LIN {X 0,Y 467.855,Z 196.206,A -85,B 0,C 180,E1 -7560,E2 -7560} C_VEL
LIN {X 0,Y 467.817,Z 196.211,A -85,B 0,C 180,E1 -7562.583,E2 -7562.583} C_VEL
LIN {X 0,Y 467.706,Z 196.227,A -85,B 0,C 180,E1 -7566.038,E2 -7566.038} C_VEL
LIN {X 0,Y 467.66,Z 196.229,A -85,B 0,C 180,E1 -7568.643,E2 -7568.643} C_VEL
LIN {X 0,Y 467.66,Z 196.234,A -85,B 0,C 180,E1 -7572.145,E2 -7572.145} C_VEL
LIN {X 0,Y 467.616,Z 196.236,A -85,B 0,C 180,E1 -7575.696,E2 -7575.696} C_VEL
LIN {X 0,Y 467.622,Z 196.233,A -85,B 0,C 180,E1 -7579.308,E2 -7579.308} C_VEL
LIN {X 0,Y 467.537,Z 196.247,A -85,B 0,C 180,E1 -7582.074,E2 -7582.074} C_VEL
LIN {X 0,Y 467.562,Z 196.239,A -85,B 0,C 180,E1 -7584.89,E2 -7584.89} C_VEL
LIN {X 0,Y 467.549,Z 196.248,A -85,B 0,C 180,E1 -7587.774,E2 -7587.774} C_VEL
LIN {X 0,Y 467.568,Z 196.24,A -85,B 0,C 180,E1 -7591.044,E2 -7591.044} C_VEL
LIN {X 0,Y 467.579,Z 196.238,A -85,B 0,C 180,E1 -7594.24,E2 -7594.24} C_VEL
LIN {X 0,Y 467.545,Z 196.245,A -85,B 0,C 180,E1 -7597.185,E2 -7597.185} C_VEL
LIN {X 0,Y 467.56,Z 196.239,A -85,B 0,C 180,E1 -7600.267,E2 -7600.267} C_VEL
LIN {X 0,Y 467.547,Z 196.244,A -85,B 0,C 180,E1 -7603.746,E2 -7603.746} C_VEL
LIN {X 0,Y 467.547,Z 196.241,A -85,B 0,C 180,E1 -7606.254,E2 -7606.254} C_VEL
LIN {X 0,Y 467.559,Z 196.241,A -85,B 0,C 180,E1 -7609.733,E2 -7609.733} C_VEL
LIN {X 0,Y 467.545,Z 196.245,A -85,B 0,C 180,E1 -7612.815,E2 -7612.815} C_VEL
LIN {X 0,Y 467.578,Z 196.237,A -85,B 0,C 180,E1 -7615.76,E2 -7615.76} C_VEL
LIN {X 0,Y 467.55,Z 196.248,A -85,B 0,C 180,E1 -7618.959,E2 -7618.959} C_VEL
LIN {X 0,Y 467.613,Z 196.32,A -85,B 0,C 180,E1 -7622.23,E2 -7622.23} C_VEL
LIN {X 0,Y 470.285,Z 209.821,A -85,B 0,C 180,E1 -7624.555,E2 -7624.555} C_VEL
LIN {X 0,Y 469.734,Z 224.485,A -85,B 0,C 180,E1 -7626.874,E2 -7626.874} C_VEL
LIN {X 0,Y 468.948,Z 244.938,A -85,B 0,C 180,E1 -7630.065,E2 -7630.065} C_VEL
LIN {X 0,Y 468.232,Z 264.095,A -85,B 0,C 180,E1 -7633.005,E2 -7633.005} C_VEL
LIN {X 0,Y 471.04,Z 286.598,A -85,B 0,C 180,E1 -7633.47,E2 -7633.47} C_VEL
LIN {X 0,Y 470.274,Z 373.12,A -85,B 0,C 180,E1 -7634.867,E2 -7634.867} C_VEL
LIN {X 0,Y 469.84,Z 386.276,A -85,B 0,C 180,E1 -7635.24,E2 -7635.24} C_VEL
LIN {X 0,Y 469.395,Z 399.568,A -85,B 0,C 180,E1 -7635.808,E2 -7635.808} C_VEL
LIN {X 0,Y 468.88,Z 410.763,A -85,B 0,C 180,E1 -7636.455,E2 -7636.455} C_VEL
LIN {X 0,Y 468.297,Z 422.997,A -85,B 0,C 180,E1 -7637.369,E2 -7637.369} C_VEL
LIN {X 0,Y 467.927,Z 434.003,A -85,B 0,C 180,E1 -7638.411,E2 -7638.411} C_VEL
LIN {X 0,Y 467.422,Z 444.065,A -85,B 0,C 180,E1 -7639.605,E2 -7639.605} C_VEL
LIN {X 0,Y 467.139,Z 452.942,A -85,B 0,C 180,E1 -7640.911,E2 -7640.911} C_VEL
LIN {X 0,Y 466.928,Z 460.016,A -85,B 0,C 180,E1 -7642.214,E2 -7642.214} C_VEL
LIN {X 0,Y 466.829,Z 465.703,A -85,B 0,C 180,E1 -7643.523,E2 -7643.523} C_VEL
LIN {X 0,Y 466.765,Z 470.118,A -85,B 0,C 180,E1 -7644.817,E2 -7644.817} C_VEL
LIN {X 0,Y 466.697,Z 472.456,A -85,B 0,C 180,E1 -7645.682,E2 -7645.682} C_VEL
LIN {X 0,Y 466.786,Z 474.366,A -85,B 0,C 180,E1 -7646.547,E2 -7646.547} C_VEL
LIN {X 0,Y 466.787,Z 475.795,A -85,B 0,C 180,E1 -7647.411,E2 -7647.411} C_VEL
LIN {X 0,Y 466.705,Z 476.796,A -85,B 0,C 180,E1 -7648.274,E2 -7648.274} C_VEL
LIN {X 0,Y 466.651,Z 477.608,A -85,B 0,C 180,E1 -7650,E2 -7650} C_VEL
LIN {X 0,Y 466.653,Z 477.372,A -85,B 0,C 180,E1 -7650.863,E2 -7650.863} C_VEL
LIN {X 0,Y 466.706,Z 476.732,A -85,B 0,C 180,E1 -7651.726,E2 -7651.726} C_VEL
LIN {X 0,Y 466.79,Z 475.696,A -85,B 0,C 180,E1 -7652.589,E2 -7652.589} C_VEL
LIN {X 0,Y 466.8,Z 474.243,A -85,B 0,C 180,E1 -7653.452,E2 -7653.452} C_VEL
LIN {X 0,Y 466.707,Z 471.192,A -85,B 0,C 180,E1 -7654.751,E2 -7654.751} C_VEL
LIN {X 0,Y 466.747,Z 467.084,A -85,B 0,C 180,E1 -7656.05,E2 -7656.05} C_VEL
LIN {X 0,Y 466.903,Z 460.778,A -85,B 0,C 180,E1 -7657.568,E2 -7657.568} C_VEL
LIN {X 0,Y 467.063,Z 453.902,A -85,B 0,C 180,E1 -7658.872,E2 -7658.872} C_VEL
LIN {X 0,Y 467.351,Z 445.386,A -85,B 0,C 180,E1 -7660.177,E2 -7660.177} C_VEL
LIN {X 0,Y 467.801,Z 436.641,A -85,B 0,C 180,E1 -7661.262,E2 -7661.262} C_VEL
LIN {X 0,Y 468.157,Z 426.895,A -85,B 0,C 180,E1 -7662.257,E2 -7662.257} C_VEL
LIN {X 0,Y 468.706,Z 415.217,A -85,B 0,C 180,E1 -7663.218,E2 -7663.218} C_VEL
LIN {X 0,Y 469.206,Z 403.457,A -85,B 0,C 180,E1 -7663.977,E2 -7663.977} C_VEL
LIN {X 0,Y 469.675,Z 391.29,A -85,B 0,C 180,E1 -7664.57,E2 -7664.57} C_VEL
LIN {X 0,Y 470.121,Z 378.153,A -85,B 0,C 180,E1 -7665.027,E2 -7665.027} C_VEL
LIN {X 0,Y 470.426,Z 365.707,A -85,B 0,C 180,E1 -7665.294,E2 -7665.294} C_VEL
LIN {X 0,Y 470.993,Z 284.423,A -85,B 0,C 180,E1 -7666.606,E2 -7666.606} C_VEL
LIN {X 0,Y 468.16,Z 262.297,A -85,B 0,C 180,E1 -7667.094,E2 -7667.094} C_VEL
LIN {X 0,Y 468.769,Z 243.285,A -85,B 0,C 180,E1 -7669.942,E2 -7669.942} C_VEL
LIN {X 0,Y 469.439,Z 222.22,A -85,B 0,C 180,E1 -7673.141,E2 -7673.141} C_VEL
LIN {X 0,Y 469.889,Z 208.581,A -85,B 0,C 180,E1 -7675.231,E2 -7675.231} C_VEL
LIN {X 0,Y 467.93,Z 197.894,A -85,B 0,C 180,E1 -7677,E2 -7677} C_VEL
LIN {X 0,Y 467.605,Z 196.242,A -85,B 0,C 180,E1 -7677.29,E2 -7677.29} C_VEL
LIN {X 0,Y 467.564,Z 196.247,A -85,B 0,C 180,E1 -7680.734,E2 -7680.734} C_VEL
LIN {X 0,Y 467.57,Z 196.241,A -85,B 0,C 180,E1 -7683.789,E2 -7683.789} C_VEL
LIN {X 0,Y 467.524,Z 196.25,A -85,B 0,C 180,E1 -7686.962,E2 -7686.962} C_VEL
LIN {X 0,Y 467.564,Z 196.24,A -85,B 0,C 180,E1 -7689.951,E2 -7689.951} C_VEL
LIN {X 0,Y 467.56,Z 196.245,A -85,B 0,C 180,E1 -7692.563,E2 -7692.563} C_VEL
LIN {X 0,Y 467.565,Z 196.241,A -85,B 0,C 180,E1 -7695.052,E2 -7695.052} C_VEL
LIN {X 0,Y 467.567,Z 196.245,A -85,B 0,C 180,E1 -7698.596,E2 -7698.596} C_VEL
LIN {X 0,Y 467.561,Z 196.243,A -85,B 0,C 180,E1 -7701.955,E2 -7701.955} C_VEL
LIN {X 0,Y 467.562,Z 196.239,A -85,B 0,C 180,E1 -7705.167,E2 -7705.167} C_VEL
LIN {X 0,Y 467.582,Z 196.242,A -85,B 0,C 180,E1 -7708.26,E2 -7708.26} C_VEL
LIN {X 0,Y 467.555,Z 196.24,A -85,B 0,C 180,E1 -7711.249,E2 -7711.249} C_VEL
LIN {X 0,Y 467.583,Z 196.242,A -85,B 0,C 180,E1 -7714.158,E2 -7714.158} C_VEL
LIN {X 0,Y 467.576,Z 196.237,A -85,B 0,C 180,E1 -7716.996,E2 -7716.996} C_VEL
LIN {X 0,Y 467.622,Z 196.236,A -85,B 0,C 180,E1 -7719.777,E2 -7719.777} C_VEL
LIN {X 0,Y 467.594,Z 196.235,A -85,B 0,C 180,E1 -7722.506,E2 -7722.506} C_VEL
LIN {X 0,Y 467.601,Z 196.236,A -85,B 0,C 180,E1 -7725.196,E2 -7725.196} C_VEL
LIN {X 0,Y 467.656,Z 196.231,A -85,B 0,C 180,E1 -7727.854,E2 -7727.854} C_VEL
LIN {X 0,Y 467.68,Z 196.228,A -85,B 0,C 180,E1 -7731.357,E2 -7731.357} C_VEL
LIN {X 0,Y 467.735,Z 196.221,A -85,B 0,C 180,E1 -7733.962,E2 -7733.962} C_VEL
LIN {X 0,Y 467.859,Z 196.21,A -85,B 0,C 180,E1 -7737.417,E2 -7737.417} C_VEL
LIN {X 0,Y 467.882,Z 196.202,A -85,B 0,C 180,E1 -7740,E2 -7740} C_VEL
LIN {X 0,Y 467.859,Z 196.205,A -85,B 0,C 180,E1 -7742.583,E2 -7742.583} C_VEL
LIN {X 0,Y 467.724,Z 196.22,A -85,B 0,C 180,E1 -7746.038,E2 -7746.038} C_VEL
LIN {X 0,Y 467.66,Z 196.233,A -85,B 0,C 180,E1 -7749.515,E2 -7749.515} C_VEL
LIN {X 0,Y 467.654,Z 196.233,A -85,B 0,C 180,E1 -7752.358,E2 -7752.358} C_VEL
LIN {X 0,Y 467.649,Z 196.233,A -85,B 0,C 180,E1 -7755.885,E2 -7755.885} C_VEL
LIN {X 0,Y 467.628,Z 196.237,A -85,B 0,C 180,E1 -7759.308,E2 -7759.308} C_VEL
LIN {X 0,Y 467.664,Z 196.309,A -85,B 0,C 180,E1 -7760.393,E2 -7760.393} C_VEL
LIN {X 0,Y 468.236,Z 199.2,A -85,B 0,C 180,E1 -7760.97,E2 -7760.97} C_VEL
LIN {X 0,Y 470.703,Z 207.594,A -85,B 0,C 180,E1 -7761.225,E2 -7761.225} C_VEL
LIN {X 0,Y 471.622,Z 212.53,A -85,B 0,C 180,E1 -7761.345,E2 -7761.345} C_VEL
LIN {X 0,Y 470.638,Z 307.216,A -85,B 0,C 180,E1 -7762.904,E2 -7762.904} C_VEL
LIN {X 0,Y 470.441,Z 320.163,A -85,B 0,C 180,E1 -7763.292,E2 -7763.292} C_VEL
LIN {X 0,Y 470.108,Z 333.13,A -85,B 0,C 180,E1 -7763.864,E2 -7763.864} C_VEL
LIN {X 0,Y 469.705,Z 344.998,A -85,B 0,C 180,E1 -7764.58,E2 -7764.58} C_VEL
LIN {X 0,Y 469.182,Z 356.975,A -85,B 0,C 180,E1 -7765.509,E2 -7765.509} C_VEL
LIN {X 0,Y 468.735,Z 367.183,A -85,B 0,C 180,E1 -7766.516,E2 -7766.516} C_VEL
LIN {X 0,Y 468.292,Z 377.042,A -85,B 0,C 180,E1 -7767.726,E2 -7767.726} C_VEL
LIN {X 0,Y 467.817,Z 385.718,A -85,B 0,C 180,E1 -7769.055,E2 -7769.055} C_VEL
LIN {X 0,Y 467.469,Z 393.089,A -85,B 0,C 180,E1 -7770.491,E2 -7770.491} C_VEL
LIN {X 0,Y 467.257,Z 398.252,A -85,B 0,C 180,E1 -7771.765,E2 -7771.765} C_VEL
LIN {X 0,Y 467.021,Z 403.063,A -85,B 0,C 180,E1 -7773.317,E2 -7773.317} C_VEL
LIN {X 0,Y 466.843,Z 406.389,A -85,B 0,C 180,E1 -7774.894,E2 -7774.894} C_VEL
LIN {X 0,Y 466.758,Z 407.877,A -85,B 0,C 180,E1 -7775.96,E2 -7775.96} C_VEL
LIN {X 0,Y 466.714,Z 408.708,A -85,B 0,C 180,E1 -7777.051,E2 -7777.051} C_VEL
LIN {X 0,Y 466.711,Z 408.872,A -85,B 0,C 180,E1 -7778.46,E2 -7778.46} C_VEL
LIN {X 0,Y 466.727,Z 408.015,A -85,B 0,C 180,E1 -7779.829,E2 -7779.829} C_VEL
LIN {X 0,Y 466.827,Z 405.646,A -85,B 0,C 180,E1 -7781.484,E2 -7781.484} C_VEL
LIN {X 0,Y 467.062,Z 401.512,A -85,B 0,C 180,E1 -7783.189,E2 -7783.189} C_VEL
LIN {X 0,Y 467.269,Z 396.435,A -85,B 0,C 180,E1 -7784.68,E2 -7784.68} C_VEL
LIN {X 0,Y 467.486,Z 389.628,A -85,B 0,C 180,E1 -7786.188,E2 -7786.188} C_VEL
LIN {X 0,Y 467.855,Z 382.299,A -85,B 0,C 180,E1 -7787.47,E2 -7787.47} C_VEL
LIN {X 0,Y 468.317,Z 373.785,A -85,B 0,C 180,E1 -7788.677,E2 -7788.677} C_VEL
LIN {X 0,Y 468.706,Z 364.825,A -85,B 0,C 180,E1 -7789.712,E2 -7789.712} C_VEL
LIN {X 0,Y 469.123,Z 353.914,A -85,B 0,C 180,E1 -7790.732,E2 -7790.732} C_VEL
LIN {X 0,Y 469.633,Z 342.07,A -85,B 0,C 180,E1 -7791.608,E2 -7791.608} C_VEL
LIN {X 0,Y 470.004,Z 330.609,A -85,B 0,C 180,E1 -7792.26,E2 -7792.26} C_VEL
LIN {X 0,Y 470.257,Z 317.363,A -85,B 0,C 180,E1 -7792.819,E2 -7792.819} C_VEL
LIN {X 0,Y 470.415,Z 311.813,A -85,B 0,C 180,E1 -7792.992,E2 -7792.992} C_VEL
LIN {X 0,Y 469.918,Z 306.092,A -85,B 0,C 180,E1 -7793.162,E2 -7793.162} C_VEL
LIN {X 0,Y 464.426,Z 287.452,A -85,B 0,C 180,E1 -7793.665,E2 -7793.665} C_VEL
LIN {X 0,Y 463.873,Z 281.633,A -85,B 0,C 180,E1 -7793.774,E2 -7793.774} C_VEL
LIN {X 0,Y 464.524,Z 212.332,A -85,B 0,C 180,E1 -7794.906,E2 -7794.906} C_VEL
LIN {X 0,Y 462.194,Z 202.993,A -85,B 0,C 180,E1 -7795.149,E2 -7795.149} C_VEL
LIN {X 0,Y 460.908,Z 198.824,A -85,B 0,C 180,E1 -7795.279,E2 -7795.279} C_VEL
LIN {X 0,Y 460.571,Z 197.117,A -85,B 0,C 180,E1 -7795.692,E2 -7795.692} C_VEL
LIN {X 0,Y 460.537,Z 197.119,A -85,B 0,C 180,E1 -7798.745,E2 -7798.745} C_VEL
LIN {X 0,Y 460.577,Z 197.109,A -85,B 0,C 180,E1 -7802.255,E2 -7802.255} C_VEL
LIN {X 0,Y 460.529,Z 197.118,A -85,B 0,C 180,E1 -7804.704,E2 -7804.704} C_VEL
LIN {X 0,Y 460.511,Z 197.119,A -85,B 0,C 180,E1 -7807.572,E2 -7807.572} C_VEL
LIN {X 0,Y 460.568,Z 197.112,A -85,B 0,C 180,E1 -7810.385,E2 -7810.385} C_VEL
LIN {X 0,Y 460.605,Z 197.106,A -85,B 0,C 180,E1 -7814.059,E2 -7814.059} C_VEL
LIN {X 0,Y 460.611,Z 197.105,A -85,B 0,C 180,E1 -7817.666,E2 -7817.666} C_VEL
LIN {X 0,Y 460.62,Z 197.106,A -85,B 0,C 180,E1 -7821.224,E2 -7821.224} C_VEL
LIN {X 0,Y 460.688,Z 197.096,A -85,B 0,C 180,E1 -7823.87,E2 -7823.87} C_VEL
LIN {X 0,Y 460.793,Z 197.082,A -85,B 0,C 180,E1 -7827.378,E2 -7827.378} C_VEL
LIN {X 0,Y 460.851,Z 197.077,A -85,B 0,C 180,E1 -7830,E2 -7830} C_VEL
LIN {X 0,Y 460.789,Z 197.088,A -85,B 0,C 180,E1 -7832.623,E2 -7832.623} C_VEL
LIN {X 0,Y 460.687,Z 197.1,A -85,B 0,C 180,E1 -7836.13,E2 -7836.13} C_VEL
LIN {X 0,Y 460.622,Z 197.106,A -85,B 0,C 180,E1 -7838.777,E2 -7838.777} C_VEL
LIN {X 0,Y 460.611,Z 197.111,A -85,B 0,C 180,E1 -7842.334,E2 -7842.334} C_VEL
LIN {X 0,Y 460.603,Z 197.112,A -85,B 0,C 180,E1 -7845.998,E2 -7845.998} C_VEL
LIN {X 0,Y 460.569,Z 197.113,A -85,B 0,C 180,E1 -7849.616,E2 -7849.616} C_VEL
LIN {X 0,Y 460.512,Z 197.12,A -85,B 0,C 180,E1 -7852.429,E2 -7852.429} C_VEL
LIN {X 0,Y 460.549,Z 197.119,A -85,B 0,C 180,E1 -7855.797,E2 -7855.797} C_VEL
LIN {X 0,Y 460.528,Z 197.118,A -85,B 0,C 180,E1 -7858.235,E2 -7858.235} C_VEL
LIN {X 0,Y 460.522,Z 197.118,A -85,B 0,C 180,E1 -7861.283,E2 -7861.283} C_VEL
LIN {X 0,Y 460.533,Z 197.115,A -85,B 0,C 180,E1 -7864.505,E2 -7864.505} C_VEL
LIN {X 0,Y 460.5,Z 197.127,A -85,B 0,C 180,E1 -7867.624,E2 -7867.624} C_VEL
LIN {X 0,Y 460.522,Z 197.118,A -85,B 0,C 180,E1 -7871.013,E2 -7871.013} C_VEL
LIN {X 0,Y 460.508,Z 197.118,A -85,B 0,C 180,E1 -7874.169,E2 -7874.169} C_VEL
LIN {X 0,Y 460.494,Z 197.124,A -85,B 0,C 180,E1 -7877.103,E2 -7877.103} C_VEL
LIN {X 0,Y 460.515,Z 197.117,A -85,B 0,C 180,E1 -7880.136,E2 -7880.136} C_VEL
LIN {X 0,Y 460.477,Z 197.126,A -85,B 0,C 180,E1 -7883.471,E2 -7883.471} C_VEL
LIN {X 0,Y 460.522,Z 197.118,A -85,B 0,C 180,E1 -7886.675,E2 -7886.675} C_VEL
LIN {X 0,Y 460.507,Z 197.119,A -85,B 0,C 180,E1 -7889.76,E2 -7889.76} C_VEL
LIN {X 0,Y 460.52,Z 197.121,A -85,B 0,C 180,E1 -7892.753,E2 -7892.753} C_VEL
LIN {X 0,Y 460.524,Z 197.116,A -85,B 0,C 180,E1 -7895.667,E2 -7895.667} C_VEL
LIN {X 0,Y 460.525,Z 197.12,A -85,B 0,C 180,E1 -7898.578,E2 -7898.578} C_VEL
LIN {X 0,Y 460.588,Z 197.11,A -85,B 0,C 180,E1 -7901.311,E2 -7901.311} C_VEL
LIN {X 0,Y 460.608,Z 197.106,A -85,B 0,C 180,E1 -7904.059,E2 -7904.059} C_VEL
LIN {X 0,Y 460.613,Z 197.105,A -85,B 0,C 180,E1 -7907.666,E2 -7907.666} C_VEL
LIN {X 0,Y 460.62,Z 197.105,A -85,B 0,C 180,E1 -7911.224,E2 -7911.224} C_VEL
LIN {X 0,Y 460.68,Z 197.097,A -85,B 0,C 180,E1 -7913.87,E2 -7913.87} C_VEL
LIN {X 0,Y 460.792,Z 197.082,A -85,B 0,C 180,E1 -7917.378,E2 -7917.378} C_VEL
LIN {X 0,Y 460.825,Z 197.082,A -85,B 0,C 180,E1 -7920,E2 -7920} C_VEL
LIN {X 0,Y 460.761,Z 197.09,A -85,B 0,C 180,E1 -7922.623,E2 -7922.623} C_VEL
LIN {X 0,Y 460.672,Z 197.104,A -85,B 0,C 180,E1 -7926.13,E2 -7926.13} C_VEL
LIN {X 0,Y 460.613,Z 197.106,A -85,B 0,C 180,E1 -7928.777,E2 -7928.777} C_VEL
LIN {X 0,Y 460.613,Z 197.109,A -85,B 0,C 180,E1 -7932.334,E2 -7932.334} C_VEL
LIN {X 0,Y 460.56,Z 197.119,A -85,B 0,C 180,E1 -7935.978,E2 -7935.978} C_VEL
LIN {X 0,Y 460.568,Z 197.114,A -85,B 0,C 180,E1 -7939.616,E2 -7939.616} C_VEL
LIN {X 0,Y 460.513,Z 197.118,A -85,B 0,C 180,E1 -7942.429,E2 -7942.429} C_VEL
LIN {X 0,Y 460.537,Z 197.122,A -85,B 0,C 180,E1 -7945.793,E2 -7945.793} C_VEL
LIN {X 0,Y 460.523,Z 197.118,A -85,B 0,C 180,E1 -7949.232,E2 -7949.232} C_VEL
LIN {X 0,Y 460.528,Z 197.116,A -85,B 0,C 180,E1 -7952.285,E2 -7952.285} C_VEL
LIN {X 0,Y 460.509,Z 197.125,A -85,B 0,C 180,E1 -7955.446,E2 -7955.446} C_VEL
LIN {X 0,Y 460.507,Z 197.12,A -85,B 0,C 180,E1 -7958.891,E2 -7958.891} C_VEL
LIN {X 0,Y 460.504,Z 197.123,A -85,B 0,C 180,E1 -7961.598,E2 -7961.598} C_VEL
LIN {X 0,Y 460.513,Z 197.118,A -85,B 0,C 180,E1 -7964.589,E2 -7964.589} C_VEL
LIN {X 0,Y 460.477,Z 197.123,A -85,B 0,C 180,E1 -7967.813,E2 -7967.813} C_VEL
LIN {X 0,Y 460.515,Z 197.117,A -85,B 0,C 180,E1 -7970.135,E2 -7970.135} C_VEL
LIN {X 0,Y 460.475,Z 197.125,A -85,B 0,C 180,E1 -7973.47,E2 -7973.47} C_VEL
LIN {X 0,Y 460.519,Z 197.12,A -85,B 0,C 180,E1 -7976.674,E2 -7976.674} C_VEL
LIN {X 0,Y 460.505,Z 197.121,A -85,B 0,C 180,E1 -7979.759,E2 -7979.759} C_VEL
LIN {X 0,Y 460.573,Z 197.213,A -85,B 0,C 180,E1 -7982.016,E2 -7982.016} C_VEL
LIN {X 0,Y 463.321,Z 210.721,A -85,B 0,C 180,E1 -7984.385,E2 -7984.385} C_VEL
LIN {X 0,Y 462.799,Z 225.395,A -85,B 0,C 180,E1 -7986.744,E2 -7986.744} C_VEL
LIN {X 0,Y 461.935,Z 245.844,A -85,B 0,C 180,E1 -7989.981,E2 -7989.981} C_VEL
LIN {X 0,Y 461.223,Z 263.551,A -85,B 0,C 180,E1 -7992.75,E2 -7992.75} C_VEL
LIN {X 0,Y 464.206,Z 287.22,A -85,B 0,C 180,E1 -7993.251,E2 -7993.251} C_VEL
LIN {X 0,Y 463.381,Z 373.084,A -85,B 0,C 180,E1 -7994.664,E2 -7994.664} C_VEL
LIN {X 0,Y 462.9,Z 386.835,A -85,B 0,C 180,E1 -7995.07,E2 -7995.07} C_VEL
LIN {X 0,Y 462.425,Z 399.796,A -85,B 0,C 180,E1 -7995.645,E2 -7995.645} C_VEL
LIN {X 0,Y 461.856,Z 411.61,A -85,B 0,C 180,E1 -7996.357,E2 -7996.357} C_VEL
LIN {X 0,Y 461.28,Z 423.385,A -85,B 0,C 180,E1 -7997.267,E2 -7997.267} C_VEL
LIN {X 0,Y 460.863,Z 433.342,A -85,B 0,C 180,E1 -7998.231,E2 -7998.231} C_VEL
LIN {X 0,Y 460.409,Z 443.44,A -85,B 0,C 180,E1 -7999.445,E2 -7999.445} C_VEL
LIN {X 0,Y 460.071,Z 452.338,A -85,B 0,C 180,E1 -8000.77,E2 -8000.77} C_VEL
LIN {X 0,Y 459.855,Z 459.44,A -85,B 0,C 180,E1 -8002.094,E2 -8002.094} C_VEL
LIN {X 0,Y 459.725,Z 465.644,A -85,B 0,C 180,E1 -8003.557,E2 -8003.557} C_VEL
LIN {X 0,Y 459.631,Z 470.824,A -85,B 0,C 180,E1 -8005.176,E2 -8005.176} C_VEL
LIN {X 0,Y 459.712,Z 473.831,A -85,B 0,C 180,E1 -8006.494,E2 -8006.494} C_VEL
LIN {X 0,Y 459.702,Z 475.266,A -85,B 0,C 180,E1 -8007.371,E2 -8007.371} C_VEL
LIN {X 0,Y 459.643,Z 476.271,A -85,B 0,C 180,E1 -8008.247,E2 -8008.247} C_VEL
LIN {X 0,Y 459.579,Z 477.086,A -85,B 0,C 180,E1 -8010,E2 -8010} C_VEL
LIN {X 0,Y 459.585,Z 476.852,A -85,B 0,C 180,E1 -8010.876,E2 -8010.876} C_VEL
LIN {X 0,Y 459.644,Z 476.213,A -85,B 0,C 180,E1 -8011.752,E2 -8011.752} C_VEL
LIN {X 0,Y 459.706,Z 475.174,A -85,B 0,C 180,E1 -8012.629,E2 -8012.629} C_VEL
LIN {X 0,Y 459.726,Z 473.721,A -85,B 0,C 180,E1 -8013.506,E2 -8013.506} C_VEL
LIN {X 0,Y 459.636,Z 470.667,A -85,B 0,C 180,E1 -8014.824,E2 -8014.824} C_VEL
LIN {X 0,Y 459.714,Z 465.49,A -85,B 0,C 180,E1 -8016.431,E2 -8016.431} C_VEL
LIN {X 0,Y 459.855,Z 459.204,A -85,B 0,C 180,E1 -8017.906,E2 -8017.906} C_VEL
LIN {X 0,Y 460.065,Z 452.097,A -85,B 0,C 180,E1 -8019.23,E2 -8019.23} C_VEL
LIN {X 0,Y 460.401,Z 443.206,A -85,B 0,C 180,E1 -8020.555,E2 -8020.555} C_VEL
LIN {X 0,Y 460.854,Z 433.12,A -85,B 0,C 180,E1 -8021.769,E2 -8021.769} C_VEL
LIN {X 0,Y 461.276,Z 423.284,A -85,B 0,C 180,E1 -8022.731,E2 -8022.731} C_VEL
LIN {X 0,Y 461.86,Z 411.599,A -85,B 0,C 180,E1 -8023.642,E2 -8023.642} C_VEL
LIN {X 0,Y 462.486,Z 398.949,A -85,B 0,C 180,E1 -8024.408,E2 -8024.408} C_VEL
LIN {X 0,Y 462.994,Z 386.793,A -85,B 0,C 180,E1 -8024.954,E2 -8024.954} C_VEL
LIN {X 0,Y 463.41,Z 373.517,A -85,B 0,C 180,E1 -8025.362,E2 -8025.362} C_VEL
LIN {X 0,Y 463.765,Z 346.687,A -85,B 0,C 180,E1 -8025.829,E2 -8025.829} C_VEL
LIN {X 0,Y 464.232,Z 285.452,A -85,B 0,C 180,E1 -8026.841,E2 -8026.841} C_VEL
LIN {X 0,Y 461.182,Z 261.686,A -85,B 0,C 180,E1 -8027.378,E2 -8027.378} C_VEL
LIN {X 0,Y 461.784,Z 242.801,A -85,B 0,C 180,E1 -8030.257,E2 -8030.257} C_VEL
LIN {X 0,Y 462.516,Z 223.248,A -85,B 0,C 180,E1 -8033.27,E2 -8033.27} C_VEL
LIN {X 0,Y 462.943,Z 209.585,A -85,B 0,C 180,E1 -8035.395,E2 -8035.395} C_VEL
LIN {X 0,Y 460.55,Z 197.122,A -85,B 0,C 180,E1 -8037.509,E2 -8037.509} C_VEL
LIN {X 0,Y 460.503,Z 197.125,A -85,B 0,C 180,E1 -8040.24,E2 -8040.24} C_VEL
LIN {X 0,Y 460.52,Z 197.122,A -85,B 0,C 180,E1 -8043.325,E2 -8043.325} C_VEL
LIN {X 0,Y 460.473,Z 197.127,A -85,B 0,C 180,E1 -8046.53,E2 -8046.53} C_VEL
LIN {X 0,Y 460.513,Z 197.118,A -85,B 0,C 180,E1 -8049.864,E2 -8049.864} C_VEL
LIN {X 0,Y 460.492,Z 197.124,A -85,B 0,C 180,E1 -8052.897,E2 -8052.897} C_VEL
LIN {X 0,Y 460.506,Z 197.118,A -85,B 0,C 180,E1 -8055.831,E2 -8055.831} C_VEL
LIN {X 0,Y 460.52,Z 197.118,A -85,B 0,C 180,E1 -8058.987,E2 -8058.987} C_VEL
LIN {X 0,Y 460.498,Z 197.124,A -85,B 0,C 180,E1 -8062.376,E2 -8062.376} C_VEL
LIN {X 0,Y 460.545,Z 197.114,A -85,B 0,C 180,E1 -8065.623,E2 -8065.623} C_VEL
LIN {X 0,Y 460.537,Z 197.117,A -85,B 0,C 180,E1 -8068.744,E2 -8068.744} C_VEL
LIN {X 0,Y 460.551,Z 197.118,A -85,B 0,C 180,E1 -8072.261,E2 -8072.261} C_VEL
LIN {X 0,Y 460.534,Z 197.117,A -85,B 0,C 180,E1 -8074.704,E2 -8074.704} C_VEL
LIN {X 0,Y 460.511,Z 197.12,A -85,B 0,C 180,E1 -8077.571,E2 -8077.571} C_VEL
LIN {X 0,Y 460.567,Z 197.114,A -85,B 0,C 180,E1 -8080.384,E2 -8080.384} C_VEL
LIN {X 0,Y 460.604,Z 197.11,A -85,B 0,C 180,E1 -8084.059,E2 -8084.059} C_VEL
LIN {X 0,Y 460.609,Z 197.11,A -85,B 0,C 180,E1 -8087.666,E2 -8087.666} C_VEL
LIN {X 0,Y 460.627,Z 197.106,A -85,B 0,C 180,E1 -8091.224,E2 -8091.224} C_VEL
LIN {X 0,Y 460.702,Z 197.098,A -85,B 0,C 180,E1 -8093.87,E2 -8093.87} C_VEL
LIN {X 0,Y 460.799,Z 197.089,A -85,B 0,C 180,E1 -8097.377,E2 -8097.377} C_VEL
LIN {X 0,Y 460.853,Z 197.077,A -85,B 0,C 180,E1 -8100,E2 -8100} C_VEL
LIN {X 0,Y 460.8,Z 197.085,A -85,B 0,C 180,E1 -8102.622,E2 -8102.622} C_VEL
LIN {X 0,Y 460.688,Z 197.097,A -85,B 0,C 180,E1 -8106.13,E2 -8106.13} C_VEL
LIN {X 0,Y 460.619,Z 197.109,A -85,B 0,C 180,E1 -8108.776,E2 -8108.776} C_VEL
LIN {X 0,Y 460.614,Z 197.111,A -85,B 0,C 180,E1 -8112.445,E2 -8112.445} C_VEL
LIN {X 0,Y 460.6,Z 197.112,A -85,B 0,C 180,E1 -8115.998,E2 -8115.998} C_VEL
LIN {X 0,Y 460.579,Z 197.114,A -85,B 0,C 180,E1 -8119.615,E2 -8119.615} C_VEL
LIN {X 0,Y 460.599,Z 197.116,A -85,B 0,C 180,E1 -8120.137,E2 -8120.137} C_VEL
LIN {X 0,Y 461.188,Z 199.942,A -85,B 0,C 180,E1 -8120.692,E2 -8120.692} C_VEL
LIN {X 0,Y 463.82,Z 208.08,A -85,B 0,C 180,E1 -8120.947,E2 -8120.947} C_VEL
LIN {X 0,Y 464.874,Z 212.678,A -85,B 0,C 180,E1 -8121.071,E2 -8121.071} C_VEL
LIN {X 0,Y 463.836,Z 307.878,A -85,B 0,C 180,E1 -8122.672,E2 -8122.672} C_VEL
LIN {X 0,Y 463.621,Z 321.14,A -85,B 0,C 180,E1 -8123.08,E2 -8123.08} C_VEL
LIN {X 0,Y 463.26,Z 333.713,A -85,B 0,C 180,E1 -8123.645,E2 -8123.645} C_VEL
LIN {X 0,Y 462.856,Z 345.267,A -85,B 0,C 180,E1 -8124.351,E2 -8124.351} C_VEL
LIN {X 0,Y 462.375,Z 356.055,A -85,B 0,C 180,E1 -8125.188,E2 -8125.188} C_VEL
LIN {X 0,Y 461.908,Z 366.343,A -85,B 0,C 180,E1 -8126.183,E2 -8126.183} C_VEL
LIN {X 0,Y 461.479,Z 374.808,A -85,B 0,C 180,E1 -8127.186,E2 -8127.186} C_VEL
LIN {X 0,Y 461.006,Z 383.5,A -85,B 0,C 180,E1 -8128.451,E2 -8128.451} C_VEL
LIN {X 0,Y 460.595,Z 391.331,A -85,B 0,C 180,E1 -8129.874,E2 -8129.874} C_VEL
LIN {X 0,Y 460.327,Z 397.374,A -85,B 0,C 180,E1 -8131.271,E2 -8131.271} C_VEL
LIN {X 0,Y 460.008,Z 402.485,A -85,B 0,C 180,E1 -8132.83,E2 -8132.83} C_VEL
LIN {X 0,Y 459.83,Z 406.232,A -85,B 0,C 180,E1 -8134.437,E2 -8134.437} C_VEL
LIN {X 0,Y 459.686,Z 408.355,A -85,B 0,C 180,E1 -8135.875,E2 -8135.875} C_VEL
LIN {X 0,Y 459.645,Z 409.383,A -85,B 0,C 180,E1 -8137.337,E2 -8137.337} C_VEL
LIN {X 0,Y 459.633,Z 409.281,A -85,B 0,C 180,E1 -8138.822,E2 -8138.822} C_VEL
LIN {X 0,Y 459.654,Z 408.249,A -85,B 0,C 180,E1 -8140.139,E2 -8140.139} C_VEL
LIN {X 0,Y 459.767,Z 406.216,A -85,B 0,C 180,E1 -8141.495,E2 -8141.495} C_VEL
LIN {X 0,Y 459.937,Z 403.236,A -85,B 0,C 180,E1 -8142.823,E2 -8142.823} C_VEL
LIN {X 0,Y 460.089,Z 399.328,A -85,B 0,C 180,E1 -8144.116,E2 -8144.116} C_VEL
LIN {X 0,Y 460.37,Z 393.539,A -85,B 0,C 180,E1 -8145.58,E2 -8145.58} C_VEL
LIN {X 0,Y 460.732,Z 385.963,A -85,B 0,C 180,E1 -8147.07,E2 -8147.07} C_VEL
LIN {X 0,Y 461.129,Z 378.047,A -85,B 0,C 180,E1 -8148.314,E2 -8148.314} C_VEL
LIN {X 0,Y 461.533,Z 369.847,A -85,B 0,C 180,E1 -8149.368,E2 -8149.368} C_VEL
LIN {X 0,Y 462.022,Z 359.535,A -85,B 0,C 180,E1 -8150.447,E2 -8150.447} C_VEL
LIN {X 0,Y 462.428,Z 349.329,A -85,B 0,C 180,E1 -8151.313,E2 -8151.313} C_VEL
LIN {X 0,Y 462.946,Z 337.113,A -85,B 0,C 180,E1 -8152.131,E2 -8152.131} C_VEL
LIN {X 0,Y 463.317,Z 324.702,A -85,B 0,C 180,E1 -8152.753,E2 -8152.753} C_VEL
LIN {X 0,Y 463.521,Z 313.111,A -85,B 0,C 180,E1 -8153.175,E2 -8153.175} C_VEL
LIN {X 0,Y 463.697,Z 300.029,A -85,B 0,C 180,E1 -8153.479,E2 -8153.479} C_VEL
LIN {X 0,Y 463.873,Z 281.633,A -85,B 0,C 180,E1 -8153.774,E2 -8153.774} C_VEL
LIN {X 0,Y 463.336,Z 275.824,A -85,B 0,C 180,E1 -8153.888,E2 -8153.888} C_VEL
LIN {X 0,Y 457.901,Z 257.151,A -85,B 0,C 180,E1 -8154.386,E2 -8154.386} C_VEL
LIN {X 0,Y 457.323,Z 251.343,A -85,B 0,C 180,E1 -8154.505,E2 -8154.505} C_VEL
LIN {X 0,Y 457.617,Z 212.867,A -85,B 0,C 180,E1 -8155.152,E2 -8155.152} C_VEL
LIN {X 0,Y 455.52,Z 204.811,A -85,B 0,C 180,E1 -8155.369,E2 -8155.369} C_VEL
LIN {X 0,Y 453.773,Z 199.322,A -85,B 0,C 180,E1 -8155.532,E2 -8155.532} C_VEL
LIN {X 0,Y 453.514,Z 197.995,A -85,B 0,C 180,E1 -8155.856,E2 -8155.856} C_VEL
LIN {X 0,Y 453.476,Z 198.002,A -85,B 0,C 180,E1 -8159.241,E2 -8159.241} C_VEL
LIN {X 0,Y 453.532,Z 197.987,A -85,B 0,C 180,E1 -8162.297,E2 -8162.297} C_VEL
LIN {X 0,Y 453.492,Z 197.997,A -85,B 0,C 180,E1 -8165.265,E2 -8165.265} C_VEL
LIN {X 0,Y 453.481,Z 197.994,A -85,B 0,C 180,E1 -8168.415,E2 -8168.415} C_VEL
LIN {X 0,Y 453.523,Z 197.995,A -85,B 0,C 180,E1 -8171.009,E2 -8171.009} C_VEL
LIN {X 0,Y 453.57,Z 197.982,A -85,B 0,C 180,E1 -8173.88,E2 -8173.88} C_VEL
LIN {X 0,Y 453.565,Z 197.983,A -85,B 0,C 180,E1 -8177.471,E2 -8177.471} C_VEL
LIN {X 0,Y 453.586,Z 197.983,A -85,B 0,C 180,E1 -8181.087,E2 -8181.087} C_VEL
LIN {X 0,Y 453.654,Z 197.972,A -85,B 0,C 180,E1 -8183.775,E2 -8183.775} C_VEL
LIN {X 0,Y 453.737,Z 197.962,A -85,B 0,C 180,E1 -8187.337,E2 -8187.337} C_VEL
LIN {X 0,Y 453.821,Z 197.953,A -85,B 0,C 180,E1 -8190,E2 -8190} C_VEL
LIN {X 0,Y 453.733,Z 197.967,A -85,B 0,C 180,E1 -8192.664,E2 -8192.664} C_VEL
LIN {X 0,Y 453.653,Z 197.978,A -85,B 0,C 180,E1 -8196.226,E2 -8196.226} C_VEL
LIN {X 0,Y 453.587,Z 197.981,A -85,B 0,C 180,E1 -8198.914,E2 -8198.914} C_VEL
LIN {X 0,Y 453.566,Z 197.986,A -85,B 0,C 180,E1 -8202.529,E2 -8202.529} C_VEL
LIN {X 0,Y 453.546,Z 197.992,A -85,B 0,C 180,E1 -8206.196,E2 -8206.196} C_VEL
LIN {X 0,Y 453.518,Z 197.988,A -85,B 0,C 180,E1 -8209.039,E2 -8209.039} C_VEL
LIN {X 0,Y 453.478,Z 197.999,A -85,B 0,C 180,E1 -8211.836,E2 -8211.836} C_VEL
LIN {X 0,Y 453.495,Z 197.991,A -85,B 0,C 180,E1 -8214.736,E2 -8214.736} C_VEL
LIN {X 0,Y 453.508,Z 197.996,A -85,B 0,C 180,E1 -8217.953,E2 -8217.953} C_VEL
LIN {X 0,Y 453.477,Z 197.994,A -85,B 0,C 180,E1 -8220.76,E2 -8220.76} C_VEL
LIN {X 0,Y 453.479,Z 197.998,A -85,B 0,C 180,E1 -8223.913,E2 -8223.913} C_VEL
LIN {X 0,Y 453.451,Z 197.999,A -85,B 0,C 180,E1 -8227.19,E2 -8227.19} C_VEL
LIN {X 0,Y 453.472,Z 197.994,A -85,B 0,C 180,E1 -8230.612,E2 -8230.612} C_VEL
LIN {X 0,Y 453.462,Z 197.996,A -85,B 0,C 180,E1 -8234.222,E2 -8234.222} C_VEL
LIN {X 0,Y 453.45,Z 198,A -85,B 0,C 180,E1 -8237.003,E2 -8237.003} C_VEL
LIN {X 0,Y 453.473,Z 198.001,A -85,B 0,C 180,E1 -8239.413,E2 -8239.413} C_VEL
LIN {X 0,Y 453.453,Z 197.999,A -85,B 0,C 180,E1 -8242.81,E2 -8242.81} C_VEL
LIN {X 0,Y 453.47,Z 197.994,A -85,B 0,C 180,E1 -8246.087,E2 -8246.087} C_VEL
LIN {X 0,Y 453.476,Z 198,A -85,B 0,C 180,E1 -8249.24,E2 -8249.24} C_VEL
LIN {X 0,Y 453.493,Z 197.992,A -85,B 0,C 180,E1 -8252.295,E2 -8252.295} C_VEL
LIN {X 0,Y 453.497,Z 197.995,A -85,B 0,C 180,E1 -8255.265,E2 -8255.265} C_VEL
LIN {X 0,Y 453.483,Z 197.995,A -85,B 0,C 180,E1 -8258.415,E2 -8258.415} C_VEL
LIN {X 0,Y 453.525,Z 197.993,A -85,B 0,C 180,E1 -8261.009,E2 -8261.009} C_VEL
LIN {X 0,Y 453.572,Z 197.982,A -85,B 0,C 180,E1 -8263.88,E2 -8263.88} C_VEL
LIN {X 0,Y 453.567,Z 197.983,A -85,B 0,C 180,E1 -8267.471,E2 -8267.471} C_VEL
LIN {X 0,Y 453.587,Z 197.982,A -85,B 0,C 180,E1 -8271.087,E2 -8271.087} C_VEL
LIN {X 0,Y 453.646,Z 197.973,A -85,B 0,C 180,E1 -8273.774,E2 -8273.774} C_VEL
LIN {X 0,Y 453.736,Z 197.961,A -85,B 0,C 180,E1 -8277.337,E2 -8277.337} C_VEL
LIN {X 0,Y 453.794,Z 197.957,A -85,B 0,C 180,E1 -8280,E2 -8280} C_VEL
LIN {X 0,Y 453.708,Z 197.968,A -85,B 0,C 180,E1 -8282.664,E2 -8282.664} C_VEL
LIN {X 0,Y 453.639,Z 197.981,A -85,B 0,C 180,E1 -8286.226,E2 -8286.226} C_VEL
LIN {X 0,Y 453.58,Z 197.981,A -85,B 0,C 180,E1 -8288.914,E2 -8288.914} C_VEL
LIN {X 0,Y 453.568,Z 197.985,A -85,B 0,C 180,E1 -8292.529,E2 -8292.529} C_VEL
LIN {X 0,Y 453.506,Z 197.996,A -85,B 0,C 180,E1 -8296.091,E2 -8296.091} C_VEL
LIN {X 0,Y 453.52,Z 197.988,A -85,B 0,C 180,E1 -8299.039,E2 -8299.039} C_VEL
LIN {X 0,Y 453.48,Z 198.001,A -85,B 0,C 180,E1 -8301.836,E2 -8301.836} C_VEL
LIN {X 0,Y 453.472,Z 197.994,A -85,B 0,C 180,E1 -8304.737,E2 -8304.737} C_VEL
LIN {X 0,Y 453.466,Z 198,A -85,B 0,C 180,E1 -8307.943,E2 -8307.943} C_VEL
LIN {X 0,Y 453.477,Z 197.994,A -85,B 0,C 180,E1 -8310.76,E2 -8310.76} C_VEL
LIN {X 0,Y 453.469,Z 197.998,A -85,B 0,C 180,E1 -8313.914,E2 -8313.914} C_VEL
LIN {X 0,Y 453.452,Z 198.001,A -85,B 0,C 180,E1 -8317.19,E2 -8317.19} C_VEL
LIN {X 0,Y 453.472,Z 197.994,A -85,B 0,C 180,E1 -8320.612,E2 -8320.612} C_VEL
LIN {X 0,Y 453.483,Z 197.993,A -85,B 0,C 180,E1 -8324.528,E2 -8324.528} C_VEL
LIN {X 0,Y 453.438,Z 197.999,A -85,B 0,C 180,E1 -8328.071,E2 -8328.071} C_VEL
LIN {X 0,Y 453.467,Z 197.998,A -85,B 0,C 180,E1 -8330.798,E2 -8330.798} C_VEL
LIN {X 0,Y 453.453,Z 197.997,A -85,B 0,C 180,E1 -8333.917,E2 -8333.917} C_VEL
LIN {X 0,Y 453.476,Z 198,A -85,B 0,C 180,E1 -8337.15,E2 -8337.15} C_VEL
LIN {X 0,Y 453.464,Z 197.999,A -85,B 0,C 180,E1 -8340.267,E2 -8340.267} C_VEL
LIN {X 0,Y 453.568,Z 198.163,A -85,B 0,C 180,E1 -8341.811,E2 -8341.811} C_VEL
LIN {X 0,Y 456.308,Z 211.618,A -85,B 0,C 180,E1 -8344.208,E2 -8344.208} C_VEL
LIN {X 0,Y 456.168,Z 220.435,A -85,B 0,C 180,E1 -8345.661,E2 -8345.661} C_VEL
LIN {X 0,Y 455.123,Z 242.366,A -85,B 0,C 180,E1 -8349.196,E2 -8349.196} C_VEL
LIN {X 0,Y 454.304,Z 261.437,A -85,B 0,C 180,E1 -8352.233,E2 -8352.233} C_VEL
LIN {X 0,Y 454.241,Z 263.059,A -85,B 0,C 180,E1 -8352.49,E2 -8352.49} C_VEL
LIN {X 0,Y 457.37,Z 287.754,A -85,B 0,C 180,E1 -8353.025,E2 -8353.025} C_VEL
LIN {X 0,Y 456.47,Z 372.884,A -85,B 0,C 180,E1 -8354.455,E2 -8354.455} C_VEL
LIN {X 0,Y 456.001,Z 386.534,A -85,B 0,C 180,E1 -8354.868,E2 -8354.868} C_VEL
LIN {X 0,Y 455.491,Z 398.914,A -85,B 0,C 180,E1 -8355.422,E2 -8355.422} C_VEL
LIN {X 0,Y 454.896,Z 410.818,A -85,B 0,C 180,E1 -8356.144,E2 -8356.144} C_VEL
LIN {X 0,Y 454.296,Z 422.597,A -85,B 0,C 180,E1 -8357.064,E2 -8357.064} C_VEL
LIN {X 0,Y 453.793,Z 432.658,A -85,B 0,C 180,E1 -8358.045,E2 -8358.045} C_VEL
LIN {X 0,Y 453.492,Z 441.151,A -85,B 0,C 180,E1 -8359.056,E2 -8359.056} C_VEL
LIN {X 0,Y 453.06,Z 450.352,A -85,B 0,C 180,E1 -8360.4,E2 -8360.4} C_VEL
LIN {X 0,Y 452.82,Z 457.771,A -85,B 0,C 180,E1 -8361.746,E2 -8361.746} C_VEL
LIN {X 0,Y 452.668,Z 462.789,A -85,B 0,C 180,E1 -8362.865,E2 -8362.865} C_VEL
LIN {X 0,Y 452.585,Z 467.654,A -85,B 0,C 180,E1 -8364.207,E2 -8364.207} C_VEL
LIN {X 0,Y 452.523,Z 471.369,A -85,B 0,C 180,E1 -8365.546,E2 -8365.546} C_VEL
LIN {X 0,Y 452.621,Z 473.291,A -85,B 0,C 180,E1 -8366.439,E2 -8366.439} C_VEL
LIN {X 0,Y 452.62,Z 474.735,A -85,B 0,C 180,E1 -8367.33,E2 -8367.33} C_VEL
LIN {X 0,Y 452.583,Z 475.745,A -85,B 0,C 180,E1 -8368.22,E2 -8368.22} C_VEL
LIN {X 0,Y 452.51,Z 476.564,A -85,B 0,C 180,E1 -8370,E2 -8370} C_VEL
LIN {X 0,Y 452.519,Z 476.333,A -85,B 0,C 180,E1 -8370.89,E2 -8370.89} C_VEL
LIN {X 0,Y 452.584,Z 475.694,A -85,B 0,C 180,E1 -8371.779,E2 -8371.779} C_VEL
LIN {X 0,Y 452.624,Z 474.653,A -85,B 0,C 180,E1 -8372.67,E2 -8372.67} C_VEL
LIN {X 0,Y 452.634,Z 473.2,A -85,B 0,C 180,E1 -8373.561,E2 -8373.561} C_VEL
LIN {X 0,Y 452.567,Z 470.147,A -85,B 0,C 180,E1 -8374.899,E2 -8374.899} C_VEL
LIN {X 0,Y 452.611,Z 465.478,A -85,B 0,C 180,E1 -8376.396,E2 -8376.396} C_VEL
LIN {X 0,Y 452.75,Z 459.725,A -85,B 0,C 180,E1 -8377.806,E2 -8377.806} C_VEL
LIN {X 0,Y 452.976,Z 452.846,A -85,B 0,C 180,E1 -8379.15,E2 -8379.15} C_VEL
LIN {X 0,Y 453.283,Z 444.327,A -85,B 0,C 180,E1 -8380.497,E2 -8380.497} C_VEL
LIN {X 0,Y 453.769,Z 435.592,A -85,B 0,C 180,E1 -8381.615,E2 -8381.615} C_VEL
LIN {X 0,Y 454.184,Z 426.03,A -85,B 0,C 180,E1 -8382.625,E2 -8382.625} C_VEL
LIN {X 0,Y 454.752,Z 415.652,A -85,B 0,C 180,E1 -8383.518,E2 -8383.518} C_VEL
LIN {X 0,Y 455.312,Z 404.342,A -85,B 0,C 180,E1 -8384.298,E2 -8384.298} C_VEL
LIN {X 0,Y 455.857,Z 391.708,A -85,B 0,C 180,E1 -8384.965,E2 -8384.965} C_VEL
LIN {X 0,Y 456.412,Z 378.316,A -85,B 0,C 180,E1 -8385.461,E2 -8385.461} C_VEL
LIN {X 0,Y 456.766,Z 365.363,A -85,B 0,C 180,E1 -8385.763,E2 -8385.763} C_VEL
LIN {X 0,Y 457.417,Z 285.863,A -85,B 0,C 180,E1 -8387.1,E2 -8387.1} C_VEL
LIN {X 0,Y 454.179,Z 261.119,A -85,B 0,C 180,E1 -8387.67,E2 -8387.67} C_VEL
LIN {X 0,Y 454.817,Z 243.859,A -85,B 0,C 180,E1 -8390.345,E2 -8390.345} C_VEL
LIN {X 0,Y 455.571,Z 224.255,A -85,B 0,C 180,E1 -8393.406,E2 -8393.406} C_VEL
LIN {X 0,Y 456,Z 210.609,A -85,B 0,C 180,E1 -8395.565,E2 -8395.565} C_VEL
LIN {X 0,Y 453.489,Z 198,A -85,B 0,C 180,E1 -8397.744,E2 -8397.744} C_VEL
LIN {X 0,Y 453.474,Z 198.002,A -85,B 0,C 180,E1 -8400.759,E2 -8400.759} C_VEL
LIN {X 0,Y 453.468,Z 197.997,A -85,B 0,C 180,E1 -8403.913,E2 -8403.913} C_VEL
LIN {X 0,Y 453.449,Z 198.001,A -85,B 0,C 180,E1 -8407.19,E2 -8407.19} C_VEL
LIN {X 0,Y 453.471,Z 198,A -85,B 0,C 180,E1 -8410.611,E2 -8410.611} C_VEL
LIN {X 0,Y 453.46,Z 197.999,A -85,B 0,C 180,E1 -8414.222,E2 -8414.222} C_VEL
LIN {X 0,Y 453.448,Z 197.998,A -85,B 0,C 180,E1 -8417.003,E2 -8417.003} C_VEL
LIN {X 0,Y 453.471,Z 197.994,A -85,B 0,C 180,E1 -8419.412,E2 -8419.412} C_VEL
LIN {X 0,Y 453.449,Z 198.001,A -85,B 0,C 180,E1 -8422.81,E2 -8422.81} C_VEL
LIN {X 0,Y 453.476,Z 197.998,A -85,B 0,C 180,E1 -8426.087,E2 -8426.087} C_VEL
LIN {X 0,Y 453.475,Z 197.995,A -85,B 0,C 180,E1 -8429.24,E2 -8429.24} C_VEL
LIN {X 0,Y 453.507,Z 197.994,A -85,B 0,C 180,E1 -8432.295,E2 -8432.295} C_VEL
LIN {X 0,Y 453.494,Z 197.993,A -85,B 0,C 180,E1 -8435.264,E2 -8435.264} C_VEL
LIN {X 0,Y 453.48,Z 197.996,A -85,B 0,C 180,E1 -8438.415,E2 -8438.415} C_VEL
LIN {X 0,Y 453.522,Z 197.989,A -85,B 0,C 180,E1 -8441.008,E2 -8441.008} C_VEL
LIN {X 0,Y 453.569,Z 197.989,A -85,B 0,C 180,E1 -8443.88,E2 -8443.88} C_VEL
LIN {X 0,Y 453.564,Z 197.988,A -85,B 0,C 180,E1 -8447.471,E2 -8447.471} C_VEL
LIN {X 0,Y 453.591,Z 197.981,A -85,B 0,C 180,E1 -8451.087,E2 -8451.087} C_VEL
LIN {X 0,Y 453.67,Z 197.974,A -85,B 0,C 180,E1 -8453.775,E2 -8453.775} C_VEL
LIN {X 0,Y 453.743,Z 197.967,A -85,B 0,C 180,E1 -8457.337,E2 -8457.337} C_VEL
LIN {X 0,Y 453.823,Z 197.953,A -85,B 0,C 180,E1 -8460,E2 -8460} C_VEL
LIN {X 0,Y 453.744,Z 197.964,A -85,B 0,C 180,E1 -8462.663,E2 -8462.663} C_VEL
LIN {X 0,Y 453.654,Z 197.973,A -85,B 0,C 180,E1 -8466.226,E2 -8466.226} C_VEL
LIN {X 0,Y 453.585,Z 197.987,A -85,B 0,C 180,E1 -8468.913,E2 -8468.913} C_VEL
LIN {X 0,Y 453.564,Z 197.991,A -85,B 0,C 180,E1 -8472.529,E2 -8472.529} C_VEL
LIN {X 0,Y 453.544,Z 197.992,A -85,B 0,C 180,E1 -8476.196,E2 -8476.196} C_VEL
LIN {X 0,Y 453.564,Z 198.037,A -85,B 0,C 180,E1 -8479.899,E2 -8479.899} C_VEL
LIN {X 0,Y 454.083,Z 200.439,A -85,B 0,C 180,E1 -8480.38,E2 -8480.38} C_VEL
LIN {X 0,Y 457.277,Z 209.981,A -85,B 0,C 180,E1 -8480.701,E2 -8480.701} C_VEL
LIN {X 0,Y 458.146,Z 213.825,A -85,B 0,C 180,E1 -8480.807,E2 -8480.807} C_VEL
LIN {X 0,Y 457.058,Z 308.401,A -85,B 0,C 180,E1 -8482.429,E2 -8482.429} C_VEL
LIN {X 0,Y 456.821,Z 321.475,A -85,B 0,C 180,E1 -8482.835,E2 -8482.835} C_VEL
LIN {X 0,Y 456.448,Z 333.941,A -85,B 0,C 180,E1 -8483.4,E2 -8483.4} C_VEL
LIN {X 0,Y 456.023,Z 345.409,A -85,B 0,C 180,E1 -8484.105,E2 -8484.105} C_VEL
LIN {X 0,Y 455.509,Z 356.602,A -85,B 0,C 180,E1 -8484.984,E2 -8484.984} C_VEL
LIN {X 0,Y 455.021,Z 365.41,A -85,B 0,C 180,E1 -8485.834,E2 -8485.834} C_VEL
LIN {X 0,Y 454.616,Z 374.355,A -85,B 0,C 180,E1 -8486.884,E2 -8486.884} C_VEL
LIN {X 0,Y 454.104,Z 382.844,A -85,B 0,C 180,E1 -8488.095,E2 -8488.095} C_VEL
LIN {X 0,Y 453.698,Z 390.492,A -85,B 0,C 180,E1 -8489.46,E2 -8489.46} C_VEL
LIN {X 0,Y 453.387,Z 396.366,A -85,B 0,C 180,E1 -8490.766,E2 -8490.766} C_VEL
LIN {X 0,Y 453.035,Z 401.944,A -85,B 0,C 180,E1 -8492.358,E2 -8492.358} C_VEL
LIN {X 0,Y 452.819,Z 405.974,A -85,B 0,C 180,E1 -8493.969,E2 -8493.969} C_VEL
LIN {X 0,Y 452.702,Z 407.895,A -85,B 0,C 180,E1 -8495.058,E2 -8495.058} C_VEL
LIN {X 0,Y 452.596,Z 409.189,A -85,B 0,C 180,E1 -8496.162,E2 -8496.162} C_VEL
LIN {X 0,Y 452.57,Z 409.958,A -85,B 0,C 180,E1 -8497.629,E2 -8497.629} C_VEL
LIN {X 0,Y 452.551,Z 409.667,A -85,B 0,C 180,E1 -8499.06,E2 -8499.06} C_VEL
LIN {X 0,Y 452.612,Z 408.063,A -85,B 0,C 180,E1 -8500.705,E2 -8500.705} C_VEL
LIN {X 0,Y 452.816,Z 404.757,A -85,B 0,C 180,E1 -8502.466,E2 -8502.466} C_VEL
LIN {X 0,Y 452.988,Z 401.475,A -85,B 0,C 180,E1 -8503.684,E2 -8503.684} C_VEL
LIN {X 0,Y 453.261,Z 395.985,A -85,B 0,C 180,E1 -8505.22,E2 -8505.22} C_VEL
LIN {X 0,Y 453.551,Z 388.942,A -85,B 0,C 180,E1 -8506.743,E2 -8506.743} C_VEL
LIN {X 0,Y 453.968,Z 381.61,A -85,B 0,C 180,E1 -8507.996,E2 -8507.996} C_VEL
LIN {X 0,Y 454.479,Z 372.438,A -85,B 0,C 180,E1 -8509.265,E2 -8509.265} C_VEL
LIN {X 0,Y 454.946,Z 362.717,A -85,B 0,C 180,E1 -8510.358,E2 -8510.358} C_VEL
LIN {X 0,Y 455.415,Z 352.1,A -85,B 0,C 180,E1 -8511.319,E2 -8511.319} C_VEL
LIN {X 0,Y 455.903,Z 340.625,A -85,B 0,C 180,E1 -8512.14,E2 -8512.14} C_VEL
LIN {X 0,Y 456.372,Z 328.454,A -85,B 0,C 180,E1 -8512.812,E2 -8512.812} C_VEL
LIN {X 0,Y 456.6,Z 315.736,A -85,B 0,C 180,E1 -8513.321,E2 -8513.321} C_VEL
LIN {X 0,Y 456.81,Z 302.354,A -85,B 0,C 180,E1 -8513.661,E2 -8513.661} C_VEL
LIN {X 0,Y 457.323,Z 251.343,A -85,B 0,C 180,E1 -8514.505,E2 -8514.505} C_VEL
LIN {X 0,Y 456.788,Z 245.54,A -85,B 0,C 180,E1 -8514.622,E2 -8514.622} C_VEL
LIN {X 0,Y 451.557,Z 226.846,A -85,B 0,C 180,E1 -8515.135,E2 -8515.135} C_VEL
LIN {X 0,Y 450.9,Z 221.047,A -85,B 0,C 180,E1 -8515.26,E2 -8515.26} C_VEL
LIN {X 0,Y 450.843,Z 214.134,A -85,B 0,C 180,E1 -8515.383,E2 -8515.383} C_VEL
LIN {X 0,Y 448.935,Z 206.857,A -85,B 0,C 180,E1 -8515.584,E2 -8515.584} C_VEL
LIN {X 0,Y 446.654,Z 199.742,A -85,B 0,C 180,E1 -8515.805,E2 -8515.805} C_VEL
LIN {X 0,Y 446.501,Z 198.868,A -85,B 0,C 180,E1 -8516.03,E2 -8516.03} C_VEL
LIN {X 0,Y 446.427,Z 198.874,A -85,B 0,C 180,E1 -8519.751,E2 -8519.751} C_VEL
LIN {X 0,Y 446.464,Z 198.871,A -85,B 0,C 180,E1 -8522.839,E2 -8522.839} C_VEL
LIN {X 0,Y 446.46,Z 198.868,A -85,B 0,C 180,E1 -8525.925,E2 -8525.925} C_VEL
LIN {X 0,Y 446.454,Z 198.873,A -85,B 0,C 180,E1 -8528.773,E2 -8528.773} C_VEL
LIN {X 0,Y 446.451,Z 198.869,A -85,B 0,C 180,E1 -8531.649,E2 -8531.649} C_VEL
LIN {X 0,Y 446.508,Z 198.865,A -85,B 0,C 180,E1 -8534.48,E2 -8534.48} C_VEL
LIN {X 0,Y 446.518,Z 198.862,A -85,B 0,C 180,E1 -8538.193,E2 -8538.193} C_VEL
LIN {X 0,Y 446.533,Z 198.863,A -85,B 0,C 180,E1 -8540.945,E2 -8540.945} C_VEL
LIN {X 0,Y 446.622,Z 198.847,A -85,B 0,C 180,E1 -8543.676,E2 -8543.676} C_VEL
LIN {X 0,Y 446.684,Z 198.84,A -85,B 0,C 180,E1 -8547.295,E2 -8547.295} C_VEL
LIN {X 0,Y 446.791,Z 198.828,A -85,B 0,C 180,E1 -8550,E2 -8550} C_VEL
LIN {X 0,Y 446.679,Z 198.845,A -85,B 0,C 180,E1 -8552.706,E2 -8552.706} C_VEL
LIN {X 0,Y 446.621,Z 198.855,A -85,B 0,C 180,E1 -8556.324,E2 -8556.324} C_VEL
LIN {X 0,Y 446.522,Z 198.864,A -85,B 0,C 180,E1 -8559.97,E2 -8559.97} C_VEL
LIN {X 0,Y 446.523,Z 198.862,A -85,B 0,C 180,E1 -8562.73,E2 -8562.73} C_VEL
LIN {X 0,Y 446.49,Z 198.867,A -85,B 0,C 180,E1 -8566.459,E2 -8566.459} C_VEL
LIN {X 0,Y 446.47,Z 198.867,A -85,B 0,C 180,E1 -8569.303,E2 -8569.303} C_VEL
LIN {X 0,Y 446.42,Z 198.878,A -85,B 0,C 180,E1 -8572.2,E2 -8572.2} C_VEL
LIN {X 0,Y 446.44,Z 198.871,A -85,B 0,C 180,E1 -8575.154,E2 -8575.154} C_VEL
LIN {X 0,Y 446.45,Z 198.872,A -85,B 0,C 180,E1 -8578.181,E2 -8578.181} C_VEL
LIN {X 0,Y 446.417,Z 198.875,A -85,B 0,C 180,E1 -8581.301,E2 -8581.301} C_VEL
LIN {X 0,Y 446.43,Z 198.872,A -85,B 0,C 180,E1 -8584.523,E2 -8584.523} C_VEL
LIN {X 0,Y 446.412,Z 198.876,A -85,B 0,C 180,E1 -8588.079,E2 -8588.079} C_VEL
LIN {X 0,Y 446.412,Z 198.88,A -85,B 0,C 180,E1 -8591.393,E2 -8591.393} C_VEL
LIN {X 0,Y 446.452,Z 198.872,A -85,B 0,C 180,E1 -8595.104,E2 -8595.104} C_VEL
LIN {X 0,Y 446.412,Z 198.874,A -85,B 0,C 180,E1 -8598.607,E2 -8598.607} C_VEL
LIN {X 0,Y 446.413,Z 198.874,A -85,B 0,C 180,E1 -8601.922,E2 -8601.922} C_VEL
LIN {X 0,Y 446.425,Z 198.876,A -85,B 0,C 180,E1 -8605.477,E2 -8605.477} C_VEL
LIN {X 0,Y 446.417,Z 198.876,A -85,B 0,C 180,E1 -8608.7,E2 -8608.7} C_VEL
LIN {X 0,Y 446.449,Z 198.869,A -85,B 0,C 180,E1 -8611.831,E2 -8611.831} C_VEL
LIN {X 0,Y 446.441,Z 198.876,A -85,B 0,C 180,E1 -8614.847,E2 -8614.847} C_VEL
LIN {X 0,Y 446.451,Z 198.87,A -85,B 0,C 180,E1 -8618.245,E2 -8618.245} C_VEL
LIN {X 0,Y 446.452,Z 198.869,A -85,B 0,C 180,E1 -8621.649,E2 -8621.649} C_VEL
LIN {X 0,Y 446.508,Z 198.866,A -85,B 0,C 180,E1 -8624.48,E2 -8624.48} C_VEL
LIN {X 0,Y 446.52,Z 198.863,A -85,B 0,C 180,E1 -8628.193,E2 -8628.193} C_VEL
LIN {X 0,Y 446.534,Z 198.862,A -85,B 0,C 180,E1 -8630.945,E2 -8630.945} C_VEL
LIN {X 0,Y 446.615,Z 198.848,A -85,B 0,C 180,E1 -8633.676,E2 -8633.676} C_VEL
LIN {X 0,Y 446.683,Z 198.84,A -85,B 0,C 180,E1 -8637.295,E2 -8637.295} C_VEL
LIN {X 0,Y 446.764,Z 198.833,A -85,B 0,C 180,E1 -8640,E2 -8640} C_VEL
LIN {X 0,Y 446.657,Z 198.846,A -85,B 0,C 180,E1 -8642.706,E2 -8642.706} C_VEL
LIN {X 0,Y 446.609,Z 198.855,A -85,B 0,C 180,E1 -8646.324,E2 -8646.324} C_VEL
LIN {X 0,Y 446.529,Z 198.859,A -85,B 0,C 180,E1 -8649.056,E2 -8649.056} C_VEL
LIN {X 0,Y 446.525,Z 198.86,A -85,B 0,C 180,E1 -8652.73,E2 -8652.73} C_VEL
LIN {X 0,Y 446.457,Z 198.873,A -85,B 0,C 180,E1 -8656.209,E2 -8656.209} C_VEL
LIN {X 0,Y 446.471,Z 198.868,A -85,B 0,C 180,E1 -8659.303,E2 -8659.303} C_VEL
LIN {X 0,Y 446.42,Z 198.876,A -85,B 0,C 180,E1 -8662.2,E2 -8662.2} C_VEL
LIN {X 0,Y 446.424,Z 198.873,A -85,B 0,C 180,E1 -8665.154,E2 -8665.154} C_VEL
LIN {X 0,Y 446.439,Z 198.872,A -85,B 0,C 180,E1 -8668.182,E2 -8668.182} C_VEL
LIN {X 0,Y 446.417,Z 198.877,A -85,B 0,C 180,E1 -8671.3,E2 -8671.3} C_VEL
LIN {X 0,Y 446.424,Z 198.872,A -85,B 0,C 180,E1 -8674.524,E2 -8674.524} C_VEL
LIN {X 0,Y 446.413,Z 198.875,A -85,B 0,C 180,E1 -8678.078,E2 -8678.078} C_VEL
LIN {X 0,Y 446.402,Z 198.883,A -85,B 0,C 180,E1 -8681.394,E2 -8681.394} C_VEL
LIN {X 0,Y 446.452,Z 198.874,A -85,B 0,C 180,E1 -8685.104,E2 -8685.104} C_VEL
LIN {X 0,Y 446.402,Z 198.876,A -85,B 0,C 180,E1 -8688.606,E2 -8688.606} C_VEL
LIN {X 0,Y 446.413,Z 198.874,A -85,B 0,C 180,E1 -8691.922,E2 -8691.922} C_VEL
LIN {X 0,Y 446.424,Z 198.876,A -85,B 0,C 180,E1 -8695.476,E2 -8695.476} C_VEL
LIN {X 0,Y 446.41,Z 198.88,A -85,B 0,C 180,E1 -8698.699,E2 -8698.699} C_VEL
LIN {X 0,Y 446.482,Z 198.883,A -85,B 0,C 180,E1 -8701.555,E2 -8701.555} C_VEL
LIN {X 0,Y 449.285,Z 212.478,A -85,B 0,C 180,E1 -8704.024,E2 -8704.024} C_VEL
LIN {X 0,Y 449.349,Z 218.384,A -85,B 0,C 180,E1 -8705.02,E2 -8705.02} C_VEL
LIN {X 0,Y 448.389,Z 237.403,A -85,B 0,C 180,E1 -8708.145,E2 -8708.145} C_VEL
LIN {X 0,Y 447.539,Z 256.351,A -85,B 0,C 180,E1 -8711.22,E2 -8711.22} C_VEL
LIN {X 0,Y 447.241,Z 262.591,A -85,B 0,C 180,E1 -8712.225,E2 -8712.225} C_VEL
LIN {X 0,Y 450.498,Z 288.718,A -85,B 0,C 180,E1 -8712.802,E2 -8712.802} C_VEL
LIN {X 0,Y 449.587,Z 372.659,A -85,B 0,C 180,E1 -8714.24,E2 -8714.24} C_VEL
LIN {X 0,Y 449.1,Z 386.212,A -85,B 0,C 180,E1 -8714.658,E2 -8714.658} C_VEL
LIN {X 0,Y 448.544,Z 399.044,A -85,B 0,C 180,E1 -8715.249,E2 -8715.249} C_VEL
LIN {X 0,Y 447.871,Z 411.604,A -85,B 0,C 180,E1 -8716.039,E2 -8716.039} C_VEL
LIN {X 0,Y 447.279,Z 422.96,A -85,B 0,C 180,E1 -8716.956,E2 -8716.956} C_VEL
LIN {X 0,Y 446.738,Z 432.966,A -85,B 0,C 180,E1 -8717.968,E2 -8717.968} C_VEL
LIN {X 0,Y 446.366,Z 442.145,A -85,B 0,C 180,E1 -8719.109,E2 -8719.109} C_VEL
LIN {X 0,Y 445.954,Z 451.097,A -85,B 0,C 180,E1 -8720.475,E2 -8720.475} C_VEL
LIN {X 0,Y 445.721,Z 458.262,A -85,B 0,C 180,E1 -8721.841,E2 -8721.841} C_VEL
LIN {X 0,Y 445.555,Z 464.137,A -85,B 0,C 180,E1 -8723.251,E2 -8723.251} C_VEL
LIN {X 0,Y 445.515,Z 468.458,A -85,B 0,C 180,E1 -8724.569,E2 -8724.569} C_VEL
LIN {X 0,Y 445.445,Z 470.815,A -85,B 0,C 180,E1 -8725.475,E2 -8725.475} C_VEL
LIN {X 0,Y 445.534,Z 472.743,A -85,B 0,C 180,E1 -8726.382,E2 -8726.382} C_VEL
LIN {X 0,Y 445.541,Z 474.199,A -85,B 0,C 180,E1 -8727.287,E2 -8727.287} C_VEL
LIN {X 0,Y 445.524,Z 475.215,A -85,B 0,C 180,E1 -8728.192,E2 -8728.192} C_VEL
LIN {X 0,Y 445.443,Z 476.04,A -85,B 0,C 180,E1 -8730,E2 -8730} C_VEL
LIN {X 0,Y 445.455,Z 475.816,A -85,B 0,C 180,E1 -8730.904,E2 -8730.904} C_VEL
LIN {X 0,Y 445.525,Z 475.179,A -85,B 0,C 180,E1 -8731.808,E2 -8731.808} C_VEL
LIN {X 0,Y 445.545,Z 474.136,A -85,B 0,C 180,E1 -8732.712,E2 -8732.712} C_VEL
LIN {X 0,Y 445.547,Z 472.684,A -85,B 0,C 180,E1 -8733.617,E2 -8733.617} C_VEL
LIN {X 0,Y 445.497,Z 469.631,A -85,B 0,C 180,E1 -8734.977,E2 -8734.977} C_VEL
LIN {X 0,Y 445.53,Z 465.364,A -85,B 0,C 180,E1 -8736.385,E2 -8736.385} C_VEL
LIN {X 0,Y 445.681,Z 459.212,A -85,B 0,C 180,E1 -8737.931,E2 -8737.931} C_VEL
LIN {X 0,Y 445.905,Z 452.337,A -85,B 0,C 180,E1 -8739.297,E2 -8739.297} C_VEL
LIN {X 0,Y 446.266,Z 443.827,A -85,B 0,C 180,E1 -8740.663,E2 -8740.663} C_VEL
LIN {X 0,Y 446.745,Z 434.104,A -85,B 0,C 180,E1 -8741.916,E2 -8741.916} C_VEL
LIN {X 0,Y 447.323,Z 422.99,A -85,B 0,C 180,E1 -8743.069,E2 -8743.069} C_VEL
LIN {X 0,Y 447.945,Z 412.267,A -85,B 0,C 180,E1 -8743.959,E2 -8743.959} C_VEL
LIN {X 0,Y 448.61,Z 400.095,A -85,B 0,C 180,E1 -8744.748,E2 -8744.748} C_VEL
LIN {X 0,Y 449.229,Z 387.471,A -85,B 0,C 180,E1 -8745.366,E2 -8745.366} C_VEL
LIN {X 0,Y 449.712,Z 374.231,A -85,B 0,C 180,E1 -8745.813,E2 -8745.813} C_VEL
LIN {X 0,Y 449.995,Z 357.053,A -85,B 0,C 180,E1 -8746.152,E2 -8746.152} C_VEL
LIN {X 0,Y 450.641,Z 286.346,A -85,B 0,C 180,E1 -8747.365,E2 -8747.365} C_VEL
LIN {X 0,Y 447.48,Z 262.358,A -85,B 0,C 180,E1 -8747.933,E2 -8747.933} C_VEL
LIN {X 0,Y 447.232,Z 260.403,A -85,B 0,C 180,E1 -8747.997,E2 -8747.997} C_VEL
LIN {X 0,Y 447.871,Z 243.401,A -85,B 0,C 180,E1 -8750.675,E2 -8750.675} C_VEL
LIN {X 0,Y 448.712,Z 223.799,A -85,B 0,C 180,E1 -8753.785,E2 -8753.785} C_VEL
LIN {X 0,Y 449.167,Z 213.207,A -85,B 0,C 180,E1 -8755.485,E2 -8755.485} C_VEL
LIN {X 0,Y 447.559,Z 203.956,A -85,B 0,C 180,E1 -8757.09,E2 -8757.09} C_VEL
LIN {X 0,Y 446.433,Z 198.879,A -85,B 0,C 180,E1 -8757.998,E2 -8757.998} C_VEL
LIN {X 0,Y 446.415,Z 198.88,A -85,B 0,C 180,E1 -8761.3,E2 -8761.3} C_VEL
LIN {X 0,Y 446.423,Z 198.878,A -85,B 0,C 180,E1 -8764.523,E2 -8764.523} C_VEL
LIN {X 0,Y 446.41,Z 198.876,A -85,B 0,C 180,E1 -8768.078,E2 -8768.078} C_VEL
LIN {X 0,Y 446.41,Z 198.876,A -85,B 0,C 180,E1 -8771.393,E2 -8771.393} C_VEL
LIN {X 0,Y 446.45,Z 198.871,A -85,B 0,C 180,E1 -8775.104,E2 -8775.104} C_VEL
LIN {X 0,Y 446.41,Z 198.88,A -85,B 0,C 180,E1 -8778.607,E2 -8778.607} C_VEL
LIN {X 0,Y 446.41,Z 198.877,A -85,B 0,C 180,E1 -8781.921,E2 -8781.921} C_VEL
LIN {X 0,Y 446.428,Z 198.872,A -85,B 0,C 180,E1 -8785.477,E2 -8785.477} C_VEL
LIN {X 0,Y 446.415,Z 198.877,A -85,B 0,C 180,E1 -8788.699,E2 -8788.699} C_VEL
LIN {X 0,Y 446.45,Z 198.873,A -85,B 0,C 180,E1 -8791.83,E2 -8791.83} C_VEL
LIN {X 0,Y 446.438,Z 198.872,A -85,B 0,C 180,E1 -8794.846,E2 -8794.846} C_VEL
LIN {X 0,Y 446.448,Z 198.873,A -85,B 0,C 180,E1 -8798.245,E2 -8798.245} C_VEL
LIN {X 0,Y 446.451,Z 198.875,A -85,B 0,C 180,E1 -8801.649,E2 -8801.649} C_VEL
LIN {X 0,Y 446.506,Z 198.863,A -85,B 0,C 180,E1 -8804.48,E2 -8804.48} C_VEL
LIN {X 0,Y 446.517,Z 198.861,A -85,B 0,C 180,E1 -8808.193,E2 -8808.193} C_VEL
LIN {X 0,Y 446.6,Z 198.856,A -85,B 0,C 180,E1 -8811.858,E2 -8811.858} C_VEL
LIN {X 0,Y 446.642,Z 198.846,A -85,B 0,C 180,E1 -8814.582,E2 -8814.582} C_VEL
LIN {X 0,Y 446.663,Z 198.843,A -85,B 0,C 180,E1 -8818.197,E2 -8818.197} C_VEL
LIN {X 0,Y 446.793,Z 198.829,A -85,B 0,C 180,E1 -8820,E2 -8820} C_VEL
LIN {X 0,Y 446.691,Z 198.843,A -85,B 0,C 180,E1 -8822.705,E2 -8822.705} C_VEL
LIN {X 0,Y 446.621,Z 198.849,A -85,B 0,C 180,E1 -8826.324,E2 -8826.324} C_VEL
LIN {X 0,Y 446.521,Z 198.864,A -85,B 0,C 180,E1 -8829.97,E2 -8829.97} C_VEL
LIN {X 0,Y 446.521,Z 198.87,A -85,B 0,C 180,E1 -8832.73,E2 -8832.73} C_VEL
LIN {X 0,Y 446.495,Z 198.87,A -85,B 0,C 180,E1 -8836.228,E2 -8836.228} C_VEL
LIN {X 0,Y 446.518,Z 198.999,A -85,B 0,C 180,E1 -8839.66,E2 -8839.66} C_VEL
LIN {X 0,Y 446.944,Z 200.957,A -85,B 0,C 180,E1 -8840.059,E2 -8840.059} C_VEL
LIN {X 0,Y 450.981,Z 212.676,A -85,B 0,C 180,E1 -8840.465,E2 -8840.465} C_VEL
LIN {X 0,Y 451.477,Z 216.123,A -85,B 0,C 180,E1 -8840.551,E2 -8840.551} C_VEL
LIN {X 0,Y 450.29,Z 308.405,A -85,B 0,C 180,E1 -8842.161,E2 -8842.161} C_VEL
LIN {X 0,Y 450.031,Z 321.179,A -85,B 0,C 180,E1 -8842.555,E2 -8842.555} C_VEL
LIN {X 0,Y 449.646,Z 333.74,A -85,B 0,C 180,E1 -8843.123,E2 -8843.123} C_VEL
LIN {X 0,Y 449.186,Z 346.015,A -85,B 0,C 180,E1 -8843.881,E2 -8843.881} C_VEL
LIN {X 0,Y 448.623,Z 357.601,A -85,B 0,C 180,E1 -8844.81,E2 -8844.81} C_VEL
LIN {X 0,Y 448.076,Z 367.517,A -85,B 0,C 180,E1 -8845.801,E2 -8845.801} C_VEL
LIN {X 0,Y 447.559,Z 376.646,A -85,B 0,C 180,E1 -8846.929,E2 -8846.929} C_VEL
LIN {X 0,Y 447.019,Z 385.621,A -85,B 0,C 180,E1 -8848.306,E2 -8848.306} C_VEL
LIN {X 0,Y 446.609,Z 392.459,A -85,B 0,C 180,E1 -8849.608,E2 -8849.608} C_VEL
LIN {X 0,Y 446.327,Z 397.459,A -85,B 0,C 180,E1 -8850.781,E2 -8850.781} C_VEL
LIN {X 0,Y 445.963,Z 402.899,A -85,B 0,C 180,E1 -8852.399,E2 -8852.399} C_VEL
LIN {X 0,Y 445.737,Z 406.791,A -85,B 0,C 180,E1 -8854.037,E2 -8854.037} C_VEL
LIN {X 0,Y 445.554,Z 409.323,A -85,B 0,C 180,E1 -8855.706,E2 -8855.706} C_VEL
LIN {X 0,Y 445.502,Z 410.222,A -85,B 0,C 180,E1 -8856.832,E2 -8856.832} C_VEL
LIN {X 0,Y 445.489,Z 410.531,A -85,B 0,C 180,E1 -8857.971,E2 -8857.971} C_VEL
LIN {X 0,Y 445.488,Z 410.009,A -85,B 0,C 180,E1 -8859.374,E2 -8859.374} C_VEL
LIN {X 0,Y 445.555,Z 408.507,A -85,B 0,C 180,E1 -8860.788,E2 -8860.788} C_VEL
LIN {X 0,Y 445.701,Z 406.05,A -85,B 0,C 180,E1 -8862.174,E2 -8862.174} C_VEL
LIN {X 0,Y 445.908,Z 402.642,A -85,B 0,C 180,E1 -8863.531,E2 -8863.531} C_VEL
LIN {X 0,Y 446.108,Z 398.289,A -85,B 0,C 180,E1 -8864.852,E2 -8864.852} C_VEL
LIN {X 0,Y 446.357,Z 392.91,A -85,B 0,C 180,E1 -8866.149,E2 -8866.149} C_VEL
LIN {X 0,Y 446.704,Z 386.358,A -85,B 0,C 180,E1 -8867.428,E2 -8867.428} C_VEL
LIN {X 0,Y 447.177,Z 378.355,A -85,B 0,C 180,E1 -8868.694,E2 -8868.694} C_VEL
LIN {X 0,Y 447.71,Z 368.618,A -85,B 0,C 180,E1 -8869.939,E2 -8869.939} C_VEL
LIN {X 0,Y 448.222,Z 358.238,A -85,B 0,C 180,E1 -8871.013,E2 -8871.013} C_VEL
LIN {X 0,Y 448.756,Z 346.972,A -85,B 0,C 180,E1 -8871.936,E2 -8871.936} C_VEL
LIN {X 0,Y 449.274,Z 335.287,A -85,B 0,C 180,E1 -8872.686,E2 -8872.686} C_VEL
LIN {X 0,Y 449.604,Z 323.526,A -85,B 0,C 180,E1 -8873.262,E2 -8873.262} C_VEL
LIN {X 0,Y 449.844,Z 311.689,A -85,B 0,C 180,E1 -8873.675,E2 -8873.675} C_VEL
LIN {X 0,Y 450.045,Z 297.45,A -85,B 0,C 180,E1 -8873.974,E2 -8873.974} C_VEL
LIN {X 0,Y 450.9,Z 221.047,A -85,B 0,C 180,E1 -8875.26,E2 -8875.26} C_VEL
LIN {X 0,Y 450.056,Z 217.328,A -85,B 0,C 180,E1 -8875.357,E2 -8875.357} C_VEL
LIN {X 0,Y 448.129,Z 214.007,A -85,B 0,C 180,E1 -8875.489,E2 -8875.489} C_VEL
LIN {X 0,Y 441.645,Z 205.716,A -85,B 0,C 180,E1 -8875.891,E2 -8875.891} C_VEL
LIN {X 0,Y 440.51,Z 203.317,A -85,B 0,C 180,E1 -8875.98,E2 -8875.98} C_VEL
LIN {X 0,Y 439.52,Z 200.156,A -85,B 0,C 180,E1 -8876.089,E2 -8876.089} C_VEL
LIN {X 0,Y 439.462,Z 199.744,A -85,B 0,C 180,E1 -8876.263,E2 -8876.263} C_VEL
LIN {X 0,Y 439.381,Z 199.751,A -85,B 0,C 180,E1 -8879.74,E2 -8879.74} C_VEL
LIN {X 0,Y 439.436,Z 199.743,A -85,B 0,C 180,E1 -8882.367,E2 -8882.367} C_VEL
LIN {X 0,Y 439.408,Z 199.747,A -85,B 0,C 180,E1 -8885.738,E2 -8885.738} C_VEL
LIN {X 0,Y 439.416,Z 199.746,A -85,B 0,C 180,E1 -8888.416,E2 -8888.416} C_VEL
LIN {X 0,Y 439.424,Z 199.747,A -85,B 0,C 180,E1 -8891.345,E2 -8891.345} C_VEL
LIN {X 0,Y 439.463,Z 199.74,A -85,B 0,C 180,E1 -8894.225,E2 -8894.225} C_VEL
LIN {X 0,Y 439.485,Z 199.737,A -85,B 0,C 180,E1 -8898.002,E2 -8898.002} C_VEL
LIN {X 0,Y 439.505,Z 199.734,A -85,B 0,C 180,E1 -8901.726,E2 -8901.726} C_VEL
LIN {X 0,Y 439.611,Z 199.727,A -85,B 0,C 180,E1 -8904.496,E2 -8904.496} C_VEL
LIN {X 0,Y 439.635,Z 199.721,A -85,B 0,C 180,E1 -8908.168,E2 -8908.168} C_VEL
LIN {X 0,Y 439.76,Z 199.704,A -85,B 0,C 180,E1 -8910,E2 -8910} C_VEL
LIN {X 0,Y 439.628,Z 199.722,A -85,B 0,C 180,E1 -8912.749,E2 -8912.749} C_VEL
LIN {X 0,Y 439.593,Z 199.73,A -85,B 0,C 180,E1 -8916.426,E2 -8916.426} C_VEL
LIN {X 0,Y 439.497,Z 199.735,A -85,B 0,C 180,E1 -8919.202,E2 -8919.202} C_VEL
LIN {X 0,Y 439.467,Z 199.739,A -85,B 0,C 180,E1 -8922.938,E2 -8922.938} C_VEL
LIN {X 0,Y 439.448,Z 199.746,A -85,B 0,C 180,E1 -8926.348,E2 -8926.348} C_VEL
LIN {X 0,Y 439.404,Z 199.749,A -85,B 0,C 180,E1 -8929.627,E2 -8929.627} C_VEL
LIN {X 0,Y 439.365,Z 199.753,A -85,B 0,C 180,E1 -8932.576,E2 -8932.576} C_VEL
LIN {X 0,Y 439.379,Z 199.754,A -85,B 0,C 180,E1 -8935.587,E2 -8935.587} C_VEL
LIN {X 0,Y 439.402,Z 199.747,A -85,B 0,C 180,E1 -8938.675,E2 -8938.675} C_VEL
LIN {X 0,Y 439.372,Z 199.755,A -85,B 0,C 180,E1 -8942.031,E2 -8942.031} C_VEL
LIN {X 0,Y 439.395,Z 199.751,A -85,B 0,C 180,E1 -8945.34,E2 -8945.34} C_VEL
LIN {X 0,Y 439.364,Z 199.752,A -85,B 0,C 180,E1 -8948.597,E2 -8948.597} C_VEL
LIN {X 0,Y 439.372,Z 199.755,A -85,B 0,C 180,E1 -8951.254,E2 -8951.254} C_VEL
LIN {X 0,Y 439.401,Z 199.748,A -85,B 0,C 180,E1 -8954.73,E2 -8954.73} C_VEL
LIN {X 0,Y 439.384,Z 199.752,A -85,B 0,C 180,E1 -8957.794,E2 -8957.794} C_VEL
LIN {X 0,Y 439.364,Z 199.758,A -85,B 0,C 180,E1 -8961.403,E2 -8961.403} C_VEL
LIN {X 0,Y 439.398,Z 199.751,A -85,B 0,C 180,E1 -8964.844,E2 -8964.844} C_VEL
LIN {X 0,Y 439.374,Z 199.75,A -85,B 0,C 180,E1 -8968.14,E2 -8968.14} C_VEL
LIN {X 0,Y 439.403,Z 199.748,A -85,B 0,C 180,E1 -8971.606,E2 -8971.606} C_VEL
LIN {X 0,Y 439.379,Z 199.751,A -85,B 0,C 180,E1 -8974.414,E2 -8974.414} C_VEL
LIN {X 0,Y 439.366,Z 199.753,A -85,B 0,C 180,E1 -8977.425,E2 -8977.425} C_VEL
LIN {X 0,Y 439.444,Z 199.747,A -85,B 0,C 180,E1 -8980.663,E2 -8980.663} C_VEL
LIN {X 0,Y 439.464,Z 199.741,A -85,B 0,C 180,E1 -8984.225,E2 -8984.225} C_VEL
LIN {X 0,Y 439.486,Z 199.737,A -85,B 0,C 180,E1 -8988.001,E2 -8988.001} C_VEL
LIN {X 0,Y 439.506,Z 199.734,A -85,B 0,C 180,E1 -8991.726,E2 -8991.726} C_VEL
LIN {X 0,Y 439.607,Z 199.729,A -85,B 0,C 180,E1 -8994.496,E2 -8994.496} C_VEL
LIN {X 0,Y 439.635,Z 199.722,A -85,B 0,C 180,E1 -8998.168,E2 -8998.168} C_VEL
LIN {X 0,Y 439.713,Z 199.711,A -85,B 0,C 180,E1 -9000,E2 -9000} C_VEL
LIN {X 0,Y 439.609,Z 199.724,A -85,B 0,C 180,E1 -9002.749,E2 -9002.749} C_VEL
LIN {X 0,Y 439.562,Z 199.732,A -85,B 0,C 180,E1 -9006.426,E2 -9006.426} C_VEL
LIN {X 0,Y 439.493,Z 199.736,A -85,B 0,C 180,E1 -9009.202,E2 -9009.202} C_VEL
LIN {X 0,Y 439.468,Z 199.739,A -85,B 0,C 180,E1 -9012.938,E2 -9012.938} C_VEL
LIN {X 0,Y 439.405,Z 199.75,A -85,B 0,C 180,E1 -9016.328,E2 -9016.328} C_VEL
LIN {X 0,Y 439.405,Z 199.751,A -85,B 0,C 180,E1 -9019.626,E2 -9019.626} C_VEL
LIN {X 0,Y 439.366,Z 199.752,A -85,B 0,C 180,E1 -9022.576,E2 -9022.576} C_VEL
LIN {X 0,Y 439.369,Z 199.756,A -85,B 0,C 180,E1 -9025.587,E2 -9025.587} C_VEL
LIN {X 0,Y 439.392,Z 199.748,A -85,B 0,C 180,E1 -9028.675,E2 -9028.675} C_VEL
LIN {X 0,Y 439.369,Z 199.754,A -85,B 0,C 180,E1 -9032.029,E2 -9032.029} C_VEL
LIN {X 0,Y 439.393,Z 199.753,A -85,B 0,C 180,E1 -9035.339,E2 -9035.339} C_VEL
LIN {X 0,Y 439.365,Z 199.752,A -85,B 0,C 180,E1 -9038.597,E2 -9038.597} C_VEL
LIN {X 0,Y 439.351,Z 199.753,A -85,B 0,C 180,E1 -9042.21,E2 -9042.21} C_VEL
LIN {X 0,Y 439.399,Z 199.755,A -85,B 0,C 180,E1 -9045.27,E2 -9045.27} C_VEL
LIN {X 0,Y 439.356,Z 199.758,A -85,B 0,C 180,E1 -9049.016,E2 -9049.016} C_VEL
LIN {X 0,Y 439.369,Z 199.753,A -85,B 0,C 180,E1 -9051.609,E2 -9051.609} C_VEL
LIN {X 0,Y 439.397,Z 199.752,A -85,B 0,C 180,E1 -9054.843,E2 -9054.843} C_VEL
LIN {X 0,Y 439.368,Z 199.754,A -85,B 0,C 180,E1 -9058.139,E2 -9058.139} C_VEL
LIN {X 0,Y 439.443,Z 199.762,A -85,B 0,C 180,E1 -9061.328,E2 -9061.328} C_VEL
LIN {X 0,Y 442.487,Z 214.831,A -85,B 0,C 180,E1 -9064.101,E2 -9064.101} C_VEL
LIN {X 0,Y 442.015,Z 226.567,A -85,B 0,C 180,E1 -9066.081,E2 -9066.081} C_VEL
LIN {X 0,Y 440.993,Z 247.018,A -85,B 0,C 180,E1 -9069.475,E2 -9069.475} C_VEL
LIN {X 0,Y 440.273,Z 262.012,A -85,B 0,C 180,E1 -9071.939,E2 -9071.939} C_VEL
LIN {X 0,Y 443.665,Z 289.247,A -85,B 0,C 180,E1 -9072.569,E2 -9072.569} C_VEL
LIN {X 0,Y 442.716,Z 371.163,A -85,B 0,C 180,E1 -9073.989,E2 -9073.989} C_VEL
LIN {X 0,Y 442.234,Z 385.031,A -85,B 0,C 180,E1 -9074.414,E2 -9074.414} C_VEL
LIN {X 0,Y 441.73,Z 396.994,A -85,B 0,C 180,E1 -9074.957,E2 -9074.957} C_VEL
LIN {X 0,Y 441.026,Z 409.151,A -85,B 0,C 180,E1 -9075.7,E2 -9075.7} C_VEL
LIN {X 0,Y 440.399,Z 421.06,A -85,B 0,C 180,E1 -9076.648,E2 -9076.648} C_VEL
LIN {X 0,Y 439.855,Z 431.227,A -85,B 0,C 180,E1 -9077.66,E2 -9077.66} C_VEL
LIN {X 0,Y 439.438,Z 439.799,A -85,B 0,C 180,E1 -9078.701,E2 -9078.701} C_VEL
LIN {X 0,Y 438.929,Z 449.073,A -85,B 0,C 180,E1 -9080.088,E2 -9080.088} C_VEL
LIN {X 0,Y 438.673,Z 456.546,A -85,B 0,C 180,E1 -9081.477,E2 -9081.477} C_VEL
LIN {X 0,Y 438.492,Z 463.391,A -85,B 0,C 180,E1 -9083.096,E2 -9083.096} C_VEL
LIN {X 0,Y 438.429,Z 467.893,A -85,B 0,C 180,E1 -9084.481,E2 -9084.481} C_VEL
LIN {X 0,Y 438.371,Z 470.259,A -85,B 0,C 180,E1 -9085.402,E2 -9085.402} C_VEL
LIN {X 0,Y 438.434,Z 472.191,A -85,B 0,C 180,E1 -9086.323,E2 -9086.323} C_VEL
LIN {X 0,Y 438.464,Z 473.661,A -85,B 0,C 180,E1 -9087.244,E2 -9087.244} C_VEL
LIN {X 0,Y 438.467,Z 474.683,A -85,B 0,C 180,E1 -9088.163,E2 -9088.163} C_VEL
LIN {X 0,Y 438.379,Z 475.516,A -85,B 0,C 180,E1 -9090,E2 -9090} C_VEL
LIN {X 0,Y 438.393,Z 475.299,A -85,B 0,C 180,E1 -9090.918,E2 -9090.918} C_VEL
LIN {X 0,Y 438.468,Z 474.663,A -85,B 0,C 180,E1 -9091.837,E2 -9091.837} C_VEL
LIN {X 0,Y 438.469,Z 473.622,A -85,B 0,C 180,E1 -9092.756,E2 -9092.756} C_VEL
LIN {X 0,Y 438.445,Z 472.169,A -85,B 0,C 180,E1 -9093.676,E2 -9093.676} C_VEL
LIN {X 0,Y 438.426,Z 469.122,A -85,B 0,C 180,E1 -9095.058,E2 -9095.058} C_VEL
LIN {X 0,Y 438.448,Z 465.011,A -85,B 0,C 180,E1 -9096.442,E2 -9096.442} C_VEL
LIN {X 0,Y 438.609,Z 458.711,A -85,B 0,C 180,E1 -9098.059,E2 -9098.059} C_VEL
LIN {X 0,Y 438.837,Z 451.835,A -85,B 0,C 180,E1 -9099.448,E2 -9099.448} C_VEL
LIN {X 0,Y 439.263,Z 443.339,A -85,B 0,C 180,E1 -9100.836,E2 -9100.836} C_VEL
LIN {X 0,Y 439.699,Z 434.631,A -85,B 0,C 180,E1 -9101.993,E2 -9101.993} C_VEL
LIN {X 0,Y 440.281,Z 423.73,A -85,B 0,C 180,E1 -9103.165,E2 -9103.165} C_VEL
LIN {X 0,Y 441.021,Z 411.858,A -85,B 0,C 180,E1 -9104.182,E2 -9104.182} C_VEL
LIN {X 0,Y 441.724,Z 399.728,A -85,B 0,C 180,E1 -9104.983,E2 -9104.983} C_VEL
LIN {X 0,Y 442.363,Z 387.173,A -85,B 0,C 180,E1 -9105.61,E2 -9105.61} C_VEL
LIN {X 0,Y 442.893,Z 374.185,A -85,B 0,C 180,E1 -9106.063,E2 -9106.063} C_VEL
LIN {X 0,Y 443.246,Z 359.086,A -85,B 0,C 180,E1 -9106.375,E2 -9106.375} C_VEL
LIN {X 0,Y 443.938,Z 287.22,A -85,B 0,C 180,E1 -9107.636,E2 -9107.636} C_VEL
LIN {X 0,Y 440.684,Z 262.537,A -85,B 0,C 180,E1 -9108.234,E2 -9108.234} C_VEL
LIN {X 0,Y 440.264,Z 259.805,A -85,B 0,C 180,E1 -9108.32,E2 -9108.32} C_VEL
LIN {X 0,Y 441.05,Z 241.438,A -85,B 0,C 180,E1 -9111.254,E2 -9111.254} C_VEL
LIN {X 0,Y 441.958,Z 221.853,A -85,B 0,C 180,E1 -9114.422,E2 -9114.422} C_VEL
LIN {X 0,Y 442.265,Z 214.28,A -85,B 0,C 180,E1 -9115.66,E2 -9115.66} C_VEL
LIN {X 0,Y 440.238,Z 203.499,A -85,B 0,C 180,E1 -9117.578,E2 -9117.578} C_VEL
LIN {X 0,Y 439.401,Z 199.756,A -85,B 0,C 180,E1 -9118.301,E2 -9118.301} C_VEL
LIN {X 0,Y 439.36,Z 199.76,A -85,B 0,C 180,E1 -9120.788,E2 -9120.788} C_VEL
LIN {X 0,Y 439.385,Z 199.752,A -85,B 0,C 180,E1 -9124.044,E2 -9124.044} C_VEL
LIN {X 0,Y 439.346,Z 199.76,A -85,B 0,C 180,E1 -9126.886,E2 -9126.886} C_VEL
LIN {X 0,Y 439.348,Z 199.755,A -85,B 0,C 180,E1 -9129.84,E2 -9129.84} C_VEL
LIN {X 0,Y 439.369,Z 199.755,A -85,B 0,C 180,E1 -9132.625,E2 -9132.625} C_VEL
LIN {X 0,Y 439.399,Z 199.748,A -85,B 0,C 180,E1 -9135.27,E2 -9135.27} C_VEL
LIN {X 0,Y 439.37,Z 199.755,A -85,B 0,C 180,E1 -9138.746,E2 -9138.746} C_VEL
LIN {X 0,Y 439.364,Z 199.753,A -85,B 0,C 180,E1 -9141.609,E2 -9141.609} C_VEL
LIN {X 0,Y 439.398,Z 199.749,A -85,B 0,C 180,E1 -9144.844,E2 -9144.844} C_VEL
LIN {X 0,Y 439.373,Z 199.754,A -85,B 0,C 180,E1 -9148.139,E2 -9148.139} C_VEL
LIN {X 0,Y 439.409,Z 199.748,A -85,B 0,C 180,E1 -9151.604,E2 -9151.604} C_VEL
LIN {X 0,Y 439.378,Z 199.755,A -85,B 0,C 180,E1 -9154.413,E2 -9154.413} C_VEL
LIN {X 0,Y 439.363,Z 199.753,A -85,B 0,C 180,E1 -9157.424,E2 -9157.424} C_VEL
LIN {X 0,Y 439.44,Z 199.744,A -85,B 0,C 180,E1 -9160.663,E2 -9160.663} C_VEL
LIN {X 0,Y 439.461,Z 199.742,A -85,B 0,C 180,E1 -9164.224,E2 -9164.224} C_VEL
LIN {X 0,Y 439.483,Z 199.739,A -85,B 0,C 180,E1 -9168.001,E2 -9168.001} C_VEL
LIN {X 0,Y 439.548,Z 199.734,A -85,B 0,C 180,E1 -9171.726,E2 -9171.726} C_VEL
LIN {X 0,Y 439.618,Z 199.721,A -85,B 0,C 180,E1 -9174.496,E2 -9174.496} C_VEL
LIN {X 0,Y 439.633,Z 199.719,A -85,B 0,C 180,E1 -9178.168,E2 -9178.168} C_VEL
LIN {X 0,Y 439.763,Z 199.705,A -85,B 0,C 180,E1 -9180,E2 -9180} C_VEL
LIN {X 0,Y 439.641,Z 199.722,A -85,B 0,C 180,E1 -9182.749,E2 -9182.749} C_VEL
LIN {X 0,Y 439.584,Z 199.726,A -85,B 0,C 180,E1 -9186.503,E2 -9186.503} C_VEL
LIN {X 0,Y 439.495,Z 199.742,A -85,B 0,C 180,E1 -9189.202,E2 -9189.202} C_VEL
LIN {X 0,Y 439.466,Z 199.749,A -85,B 0,C 180,E1 -9192.938,E2 -9192.938} C_VEL
LIN {X 0,Y 439.446,Z 199.747,A -85,B 0,C 180,E1 -9196.348,E2 -9196.348} C_VEL
LIN {X 0,Y 439.508,Z 199.898,A -85,B 0,C 180,E1 -9199.381,E2 -9199.381} C_VEL
LIN {X 0,Y 439.844,Z 201.567,A -85,B 0,C 180,E1 -9199.727,E2 -9199.727} C_VEL
LIN {X 0,Y 444.502,Z 214.709,A -85,B 0,C 180,E1 -9200.204,E2 -9200.204} C_VEL
LIN {X 0,Y 444.791,Z 218.14,A -85,B 0,C 180,E1 -9200.281,E2 -9200.281} C_VEL
LIN {X 0,Y 443.536,Z 308.857,A -85,B 0,C 180,E1 -9201.892,E2 -9201.892} C_VEL
LIN {X 0,Y 443.262,Z 321.972,A -85,B 0,C 180,E1 -9202.305,E2 -9202.305} C_VEL
LIN {X 0,Y 442.866,Z 334.186,A -85,B 0,C 180,E1 -9202.867,E2 -9202.867} C_VEL
LIN {X 0,Y 442.42,Z 344.904,A -85,B 0,C 180,E1 -9203.523,E2 -9203.523} C_VEL
LIN {X 0,Y 441.857,Z 356.396,A -85,B 0,C 180,E1 -9204.428,E2 -9204.428} C_VEL
LIN {X 0,Y 441.207,Z 366.967,A -85,B 0,C 180,E1 -9205.473,E2 -9205.473} C_VEL
LIN {X 0,Y 440.756,Z 375.541,A -85,B 0,C 180,E1 -9206.517,E2 -9206.517} C_VEL
LIN {X 0,Y 440.194,Z 384.257,A -85,B 0,C 180,E1 -9207.809,E2 -9207.809} C_VEL
LIN {X 0,Y 439.733,Z 391.635,A -85,B 0,C 180,E1 -9209.174,E2 -9209.174} C_VEL
LIN {X 0,Y 439.359,Z 397.35,A -85,B 0,C 180,E1 -9210.482,E2 -9210.482} C_VEL
LIN {X 0,Y 439.015,Z 402.432,A -85,B 0,C 180,E1 -9211.956,E2 -9211.956} C_VEL
LIN {X 0,Y 438.739,Z 406.622,A -85,B 0,C 180,E1 -9213.595,E2 -9213.595} C_VEL
LIN {X 0,Y 438.551,Z 409.359,A -85,B 0,C 180,E1 -9215.234,E2 -9215.234} C_VEL
LIN {X 0,Y 438.434,Z 410.717,A -85,B 0,C 180,E1 -9216.728,E2 -9216.728} C_VEL
LIN {X 0,Y 438.398,Z 411.011,A -85,B 0,C 180,E1 -9218.231,E2 -9218.231} C_VEL
LIN {X 0,Y 438.427,Z 410.098,A -85,B 0,C 180,E1 -9219.882,E2 -9219.882} C_VEL
LIN {X 0,Y 438.572,Z 407.628,A -85,B 0,C 180,E1 -9221.684,E2 -9221.684} C_VEL
LIN {X 0,Y 438.773,Z 404.8,A -85,B 0,C 180,E1 -9222.987,E2 -9222.987} C_VEL
LIN {X 0,Y 438.949,Z 401.008,A -85,B 0,C 180,E1 -9224.301,E2 -9224.301} C_VEL
LIN {X 0,Y 439.215,Z 396.22,A -85,B 0,C 180,E1 -9225.605,E2 -9225.605} C_VEL
LIN {X 0,Y 439.521,Z 390.32,A -85,B 0,C 180,E1 -9226.902,E2 -9226.902} C_VEL
LIN {X 0,Y 439.985,Z 382.531,A -85,B 0,C 180,E1 -9228.282,E2 -9228.282} C_VEL
LIN {X 0,Y 440.521,Z 373.398,A -85,B 0,C 180,E1 -9229.581,E2 -9229.581} C_VEL
LIN {X 0,Y 441.11,Z 363.129,A -85,B 0,C 180,E1 -9230.762,E2 -9230.762} C_VEL
LIN {X 0,Y 441.616,Z 352.193,A -85,B 0,C 180,E1 -9231.763,E2 -9231.763} C_VEL
LIN {X 0,Y 442.205,Z 340.279,A -85,B 0,C 180,E1 -9232.623,E2 -9232.623} C_VEL
LIN {X 0,Y 442.612,Z 329.154,A -85,B 0,C 180,E1 -9233.244,E2 -9233.244} C_VEL
LIN {X 0,Y 442.879,Z 316.395,A -85,B 0,C 180,E1 -9233.765,E2 -9233.765} C_VEL
LIN {X 0,Y 443.105,Z 302.854,A -85,B 0,C 180,E1 -9234.115,E2 -9234.115} C_VEL
LIN {X 0,Y 444.089,Z 215.399,A -85,B 0,C 180,E1 -9235.622,E2 -9235.622} C_VEL
LIN {X 0,Y 442.232,Z 208.586,A -85,B 0,C 180,E1 -9235.817,E2 -9235.817} C_VEL
LIN {X 0,Y 440.51,Z 203.317,A -85,B 0,C 180,E1 -9235.98,E2 -9235.98} C_VEL
LIN {X 0,Y 439.517,Z 201.493,A -85,B 0,C 180,E1 -9236.14,E2 -9236.14} C_VEL
LIN {X 0,Y 438.026,Z 200.241,A -85,B 0,C 180,E1 -9236.5,E2 -9236.5} C_VEL
LIN {X 0,Y 436.243,Z 200.148,A -85,B 0,C 180,E1 -9237.069,E2 -9237.069} C_VEL
LIN {X 0,Y 433.978,Z 200.565,A -85,B 0,C 180,E1 -9238.138,E2 -9238.138} C_VEL
LIN {X 0,Y 432.552,Z 200.649,A -85,B 0,C 180,E1 -9239.338,E2 -9239.338} C_VEL
LIN {X 0,Y 432.333,Z 200.628,A -85,B 0,C 180,E1 -9239.945,E2 -9239.945} C_VEL
LIN {X 0,Y 432.385,Z 200.626,A -85,B 0,C 180,E1 -9242.928,E2 -9242.928} C_VEL
LIN {X 0,Y 432.366,Z 200.623,A -85,B 0,C 180,E1 -9246.023,E2 -9246.023} C_VEL
LIN {X 0,Y 432.351,Z 200.632,A -85,B 0,C 180,E1 -9249.046,E2 -9249.046} C_VEL
LIN {X 0,Y 432.36,Z 200.624,A -85,B 0,C 180,E1 -9252.011,E2 -9252.011} C_VEL
LIN {X 0,Y 432.395,Z 200.627,A -85,B 0,C 180,E1 -9254.927,E2 -9254.927} C_VEL
LIN {X 0,Y 432.46,Z 200.612,A -85,B 0,C 180,E1 -9257.804,E2 -9257.804} C_VEL
LIN {X 0,Y 432.465,Z 200.611,A -85,B 0,C 180,E1 -9261.59,E2 -9261.59} C_VEL
LIN {X 0,Y 432.587,Z 200.601,A -85,B 0,C 180,E1 -9264.406,E2 -9264.406} C_VEL
LIN {X 0,Y 432.604,Z 200.596,A -85,B 0,C 180,E1 -9268.138,E2 -9268.138} C_VEL
LIN {X 0,Y 432.729,Z 200.58,A -85,B 0,C 180,E1 -9270,E2 -9270} C_VEL
LIN {X 0,Y 432.58,Z 200.6,A -85,B 0,C 180,E1 -9272.794,E2 -9272.794} C_VEL
LIN {X 0,Y 432.586,Z 200.596,A -85,B 0,C 180,E1 -9275.594,E2 -9275.594} C_VEL
LIN {X 0,Y 432.466,Z 200.617,A -85,B 0,C 180,E1 -9278.41,E2 -9278.41} C_VEL
LIN {X 0,Y 432.461,Z 200.619,A -85,B 0,C 180,E1 -9282.197,E2 -9282.197} C_VEL
LIN {X 0,Y 432.431,Z 200.622,A -85,B 0,C 180,E1 -9286.039,E2 -9286.039} C_VEL
LIN {X 0,Y 432.388,Z 200.622,A -85,B 0,C 180,E1 -9289.485,E2 -9289.485} C_VEL
LIN {X 0,Y 432.318,Z 200.629,A -85,B 0,C 180,E1 -9292.965,E2 -9292.965} C_VEL
LIN {X 0,Y 432.339,Z 200.627,A -85,B 0,C 180,E1 -9295.002,E2 -9295.002} C_VEL
LIN {X 0,Y 432.349,Z 200.629,A -85,B 0,C 180,E1 -9298.126,E2 -9298.126} C_VEL
LIN {X 0,Y 432.323,Z 200.632,A -85,B 0,C 180,E1 -9301.346,E2 -9301.346} C_VEL
LIN {X 0,Y 432.341,Z 200.626,A -85,B 0,C 180,E1 -9304.677,E2 -9304.677} C_VEL
LIN {X 0,Y 432.331,Z 200.629,A -85,B 0,C 180,E1 -9308.151,E2 -9308.151} C_VEL
LIN {X 0,Y 432.32,Z 200.636,A -85,B 0,C 180,E1 -9311.6,E2 -9311.6} C_VEL
LIN {X 0,Y 432.336,Z 200.627,A -85,B 0,C 180,E1 -9314.348,E2 -9314.348} C_VEL
LIN {X 0,Y 432.318,Z 200.632,A -85,B 0,C 180,E1 -9317.017,E2 -9317.017} C_VEL
LIN {X 0,Y 432.293,Z 200.634,A -85,B 0,C 180,E1 -9319.828,E2 -9319.828} C_VEL
LIN {X 0,Y 432.308,Z 200.635,A -85,B 0,C 180,E1 -9323.022,E2 -9323.022} C_VEL
LIN {X 0,Y 432.36,Z 200.624,A -85,B 0,C 180,E1 -9325.997,E2 -9325.997} C_VEL
LIN {X 0,Y 432.348,Z 200.628,A -85,B 0,C 180,E1 -9329.49,E2 -9329.49} C_VEL
LIN {X 0,Y 432.342,Z 200.627,A -85,B 0,C 180,E1 -9331.874,E2 -9331.874} C_VEL
LIN {X 0,Y 432.38,Z 200.623,A -85,B 0,C 180,E1 -9335.539,E2 -9335.539} C_VEL
LIN {X 0,Y 432.353,Z 200.63,A -85,B 0,C 180,E1 -9339.046,E2 -9339.046} C_VEL
LIN {X 0,Y 432.362,Z 200.624,A -85,B 0,C 180,E1 -9342.011,E2 -9342.011} C_VEL
LIN {X 0,Y 432.395,Z 200.625,A -85,B 0,C 180,E1 -9344.926,E2 -9344.926} C_VEL
LIN {X 0,Y 432.462,Z 200.612,A -85,B 0,C 180,E1 -9347.804,E2 -9347.804} C_VEL
LIN {X 0,Y 432.467,Z 200.611,A -85,B 0,C 180,E1 -9351.59,E2 -9351.59} C_VEL
LIN {X 0,Y 432.58,Z 200.603,A -85,B 0,C 180,E1 -9354.406,E2 -9354.406} C_VEL
LIN {X 0,Y 432.604,Z 200.598,A -85,B 0,C 180,E1 -9358.138,E2 -9358.138} C_VEL
LIN {X 0,Y 432.663,Z 200.59,A -85,B 0,C 180,E1 -9360,E2 -9360} C_VEL
LIN {X 0,Y 432.562,Z 200.601,A -85,B 0,C 180,E1 -9362.794,E2 -9362.794} C_VEL
LIN {X 0,Y 432.575,Z 200.598,A -85,B 0,C 180,E1 -9365.594,E2 -9365.594} C_VEL
LIN {X 0,Y 432.465,Z 200.616,A -85,B 0,C 180,E1 -9368.41,E2 -9368.41} C_VEL
LIN {X 0,Y 432.462,Z 200.617,A -85,B 0,C 180,E1 -9372.197,E2 -9372.197} C_VEL
LIN {X 0,Y 432.392,Z 200.627,A -85,B 0,C 180,E1 -9376.04,E2 -9376.04} C_VEL
LIN {X 0,Y 432.39,Z 200.623,A -85,B 0,C 180,E1 -9379.485,E2 -9379.485} C_VEL
LIN {X 0,Y 432.315,Z 200.63,A -85,B 0,C 180,E1 -9382.965,E2 -9382.965} C_VEL
LIN {X 0,Y 432.32,Z 200.633,A -85,B 0,C 180,E1 -9386.035,E2 -9386.035} C_VEL
LIN {X 0,Y 432.329,Z 200.63,A -85,B 0,C 180,E1 -9389.189,E2 -9389.189} C_VEL
LIN {X 0,Y 432.324,Z 200.629,A -85,B 0,C 180,E1 -9392.443,E2 -9392.443} C_VEL
LIN {X 0,Y 432.339,Z 200.631,A -85,B 0,C 180,E1 -9395.818,E2 -9395.818} C_VEL
LIN {X 0,Y 432.328,Z 200.629,A -85,B 0,C 180,E1 -9398.712,E2 -9398.712} C_VEL
LIN {X 0,Y 432.306,Z 200.633,A -85,B 0,C 180,E1 -9401.801,E2 -9401.801} C_VEL
LIN {X 0,Y 432.336,Z 200.627,A -85,B 0,C 180,E1 -9404.347,E2 -9404.347} C_VEL
LIN {X 0,Y 432.304,Z 200.636,A -85,B 0,C 180,E1 -9407.018,E2 -9407.018} C_VEL
LIN {X 0,Y 432.31,Z 200.631,A -85,B 0,C 180,E1 -9409.825,E2 -9409.825} C_VEL
LIN {X 0,Y 432.307,Z 200.637,A -85,B 0,C 180,E1 -9413.022,E2 -9413.022} C_VEL
LIN {X 0,Y 432.335,Z 200.627,A -85,B 0,C 180,E1 -9416.002,E2 -9416.002} C_VEL
LIN {X 0,Y 432.343,Z 200.631,A -85,B 0,C 180,E1 -9419.491,E2 -9419.491} C_VEL
LIN {X 0,Y 432.403,Z 200.628,A -85,B 0,C 180,E1 -9421.091,E2 -9421.091} C_VEL
LIN {X 0,Y 435.464,Z 215.665,A -85,B 0,C 180,E1 -9423.909,E2 -9423.909} C_VEL
LIN {X 0,Y 435.36,Z 223.029,A -85,B 0,C 180,E1 -9425.183,E2 -9425.183} C_VEL
LIN {X 0,Y 434.251,Z 242.018,A -85,B 0,C 180,E1 -9428.396,E2 -9428.396} C_VEL
LIN {X 0,Y 433.392,Z 259.64,A -85,B 0,C 180,E1 -9431.345,E2 -9431.345} C_VEL
LIN {X 0,Y 433.31,Z 261.792,A -85,B 0,C 180,E1 -9431.683,E2 -9431.683} C_VEL
LIN {X 0,Y 436.824,Z 289.188,A -85,B 0,C 180,E1 -9432.315,E2 -9432.315} C_VEL
LIN {X 0,Y 435.841,Z 370.736,A -85,B 0,C 180,E1 -9433.759,E2 -9433.759} C_VEL
LIN {X 0,Y 435.405,Z 383.821,A -85,B 0,C 180,E1 -9434.163,E2 -9434.163} C_VEL
LIN {X 0,Y 434.78,Z 397.081,A -85,B 0,C 180,E1 -9434.771,E2 -9434.771} C_VEL
LIN {X 0,Y 434.155,Z 408.282,A -85,B 0,C 180,E1 -9435.468,E2 -9435.468} C_VEL
LIN {X 0,Y 433.426,Z 419.95,A -85,B 0,C 180,E1 -9436.402,E2 -9436.402} C_VEL
LIN {X 0,Y 432.896,Z 430.481,A -85,B 0,C 180,E1 -9437.459,E2 -9437.459} C_VEL
LIN {X 0,Y 432.439,Z 439.095,A -85,B 0,C 180,E1 -9438.516,E2 -9438.516} C_VEL
LIN {X 0,Y 431.864,Z 448.413,A -85,B 0,C 180,E1 -9439.924,E2 -9439.924} C_VEL
LIN {X 0,Y 431.602,Z 455.915,A -85,B 0,C 180,E1 -9441.337,E2 -9441.337} C_VEL
LIN {X 0,Y 431.41,Z 462.795,A -85,B 0,C 180,E1 -9442.982,E2 -9442.982} C_VEL
LIN {X 0,Y 431.345,Z 467.318,A -85,B 0,C 180,E1 -9444.39,E2 -9444.39} C_VEL
LIN {X 0,Y 431.301,Z 469.693,A -85,B 0,C 180,E1 -9445.326,E2 -9445.326} C_VEL
LIN {X 0,Y 431.337,Z 471.632,A -85,B 0,C 180,E1 -9446.263,E2 -9446.263} C_VEL
LIN {X 0,Y 431.389,Z 473.118,A -85,B 0,C 180,E1 -9447.198,E2 -9447.198} C_VEL
LIN {X 0,Y 431.41,Z 474.148,A -85,B 0,C 180,E1 -9448.133,E2 -9448.133} C_VEL
LIN {X 0,Y 431.316,Z 474.99,A -85,B 0,C 180,E1 -9450,E2 -9450} C_VEL
LIN {X 0,Y 431.333,Z 474.783,A -85,B 0,C 180,E1 -9450.933,E2 -9450.933} C_VEL
LIN {X 0,Y 431.394,Z 474.149,A -85,B 0,C 180,E1 -9451.867,E2 -9451.867} C_VEL
LIN {X 0,Y 431.394,Z 473.109,A -85,B 0,C 180,E1 -9452.801,E2 -9452.801} C_VEL
LIN {X 0,Y 431.346,Z 471.657,A -85,B 0,C 180,E1 -9453.737,E2 -9453.737} C_VEL
LIN {X 0,Y 431.356,Z 468.616,A -85,B 0,C 180,E1 -9455.141,E2 -9455.141} C_VEL
LIN {X 0,Y 431.376,Z 464.511,A -85,B 0,C 180,E1 -9456.548,E2 -9456.548} C_VEL
LIN {X 0,Y 431.554,Z 458.224,A -85,B 0,C 180,E1 -9458.192,E2 -9458.192} C_VEL
LIN {X 0,Y 431.788,Z 451.359,A -85,B 0,C 180,E1 -9459.604,E2 -9459.604} C_VEL
LIN {X 0,Y 432.248,Z 442.868,A -85,B 0,C 180,E1 -9461.014,E2 -9461.014} C_VEL
LIN {X 0,Y 432.682,Z 434.177,A -85,B 0,C 180,E1 -9462.19,E2 -9462.19} C_VEL
LIN {X 0,Y 433.288,Z 424.213,A -85,B 0,C 180,E1 -9463.291,E2 -9463.291} C_VEL
LIN {X 0,Y 434.024,Z 412.952,A -85,B 0,C 180,E1 -9464.296,E2 -9464.296} C_VEL
LIN {X 0,Y 434.775,Z 401.43,A -85,B 0,C 180,E1 -9465.109,E2 -9465.109} C_VEL
LIN {X 0,Y 435.41,Z 389.605,A -85,B 0,C 180,E1 -9465.746,E2 -9465.746} C_VEL
LIN {X 0,Y 436.03,Z 376.141,A -85,B 0,C 180,E1 -9466.263,E2 -9466.263} C_VEL
LIN {X 0,Y 436.436,Z 363.005,A -85,B 0,C 180,E1 -9466.578,E2 -9466.578} C_VEL
LIN {X 0,Y 437.215,Z 288.095,A -85,B 0,C 180,E1 -9467.916,E2 -9467.916} C_VEL
LIN {X 0,Y 434.081,Z 264.092,A -85,B 0,C 180,E1 -9468.512,E2 -9468.512} C_VEL
LIN {X 0,Y 433.345,Z 259.175,A -85,B 0,C 180,E1 -9468.657,E2 -9468.657} C_VEL
LIN {X 0,Y 434.181,Z 241.047,A -85,B 0,C 180,E1 -9471.608,E2 -9471.608} C_VEL
LIN {X 0,Y 435.299,Z 218.634,A -85,B 0,C 180,E1 -9475.293,E2 -9475.293} C_VEL
LIN {X 0,Y 435.149,Z 213.861,A -85,B 0,C 180,E1 -9476.111,E2 -9476.111} C_VEL
LIN {X 0,Y 432.374,Z 200.633,A -85,B 0,C 180,E1 -9478.554,E2 -9478.554} C_VEL
LIN {X 0,Y 432.32,Z 200.636,A -85,B 0,C 180,E1 -9481.346,E2 -9481.346} C_VEL
LIN {X 0,Y 432.337,Z 200.634,A -85,B 0,C 180,E1 -9484.677,E2 -9484.677} C_VEL
LIN {X 0,Y 432.329,Z 200.631,A -85,B 0,C 180,E1 -9488.151,E2 -9488.151} C_VEL
LIN {X 0,Y 432.32,Z 200.63,A -85,B 0,C 180,E1 -9491.798,E2 -9491.798} C_VEL
LIN {X 0,Y 432.334,Z 200.632,A -85,B 0,C 180,E1 -9494.347,E2 -9494.347} C_VEL
LIN {X 0,Y 432.316,Z 200.63,A -85,B 0,C 180,E1 -9497.016,E2 -9497.016} C_VEL
LIN {X 0,Y 432.308,Z 200.631,A -85,B 0,C 180,E1 -9499.825,E2 -9499.825} C_VEL
LIN {X 0,Y 432.304,Z 200.634,A -85,B 0,C 180,E1 -9503.022,E2 -9503.022} C_VEL
LIN {X 0,Y 432.359,Z 200.628,A -85,B 0,C 180,E1 -9505.996,E2 -9505.996} C_VEL
LIN {X 0,Y 432.346,Z 200.628,A -85,B 0,C 180,E1 -9509.49,E2 -9509.49} C_VEL
LIN {X 0,Y 432.347,Z 200.63,A -85,B 0,C 180,E1 -9511.874,E2 -9511.874} C_VEL
LIN {X 0,Y 432.377,Z 200.626,A -85,B 0,C 180,E1 -9515.539,E2 -9515.539} C_VEL
LIN {X 0,Y 432.35,Z 200.626,A -85,B 0,C 180,E1 -9519.046,E2 -9519.046} C_VEL
LIN {X 0,Y 432.359,Z 200.627,A -85,B 0,C 180,E1 -9522.01,E2 -9522.01} C_VEL
LIN {X 0,Y 432.393,Z 200.62,A -85,B 0,C 180,E1 -9524.926,E2 -9524.926} C_VEL
LIN {X 0,Y 432.459,Z 200.615,A -85,B 0,C 180,E1 -9527.803,E2 -9527.803} C_VEL
LIN {X 0,Y 432.492,Z 200.612,A -85,B 0,C 180,E1 -9531.59,E2 -9531.59} C_VEL
LIN {X 0,Y 432.594,Z 200.597,A -85,B 0,C 180,E1 -9534.406,E2 -9534.406} C_VEL
LIN {X 0,Y 432.603,Z 200.595,A -85,B 0,C 180,E1 -9538.138,E2 -9538.138} C_VEL
LIN {X 0,Y 432.732,Z 200.581,A -85,B 0,C 180,E1 -9540,E2 -9540} C_VEL
LIN {X 0,Y 432.592,Z 200.6,A -85,B 0,C 180,E1 -9542.794,E2 -9542.794} C_VEL
LIN {X 0,Y 432.543,Z 200.604,A -85,B 0,C 180,E1 -9546.504,E2 -9546.504} C_VEL
LIN {X 0,Y 432.439,Z 200.621,A -85,B 0,C 180,E1 -9549.353,E2 -9549.353} C_VEL
LIN {X 0,Y 432.431,Z 200.626,A -85,B 0,C 180,E1 -9552.804,E2 -9552.804} C_VEL
LIN {X 0,Y 432.412,Z 200.624,A -85,B 0,C 180,E1 -9556.479,E2 -9556.479} C_VEL
LIN {X 0,Y 432.454,Z 200.798,A -85,B 0,C 180,E1 -9559.089,E2 -9559.089} C_VEL
LIN {X 0,Y 432.785,Z 202.213,A -85,B 0,C 180,E1 -9559.388,E2 -9559.388} C_VEL
LIN {X 0,Y 437.993,Z 216.487,A -85,B 0,C 180,E1 -9559.927,E2 -9559.927} C_VEL
LIN {X 0,Y 436.792,Z 309.757,A -85,B 0,C 180,E1 -9561.627,E2 -9561.627} C_VEL
LIN {X 0,Y 436.513,Z 321.963,A -85,B 0,C 180,E1 -9562.014,E2 -9562.014} C_VEL
LIN {X 0,Y 436.084,Z 335.147,A -85,B 0,C 180,E1 -9562.63,E2 -9562.63} C_VEL
LIN {X 0,Y 435.539,Z 347.09,A -85,B 0,C 180,E1 -9563.392,E2 -9563.392} C_VEL
LIN {X 0,Y 434.941,Z 358.492,A -85,B 0,C 180,E1 -9564.333,E2 -9564.333} C_VEL
LIN {X 0,Y 434.293,Z 369.143,A -85,B 0,C 180,E1 -9565.436,E2 -9565.436} C_VEL
LIN {X 0,Y 433.637,Z 378.825,A -85,B 0,C 180,E1 -9566.696,E2 -9566.696} C_VEL
LIN {X 0,Y 433.06,Z 387.378,A -85,B 0,C 180,E1 -9568.075,E2 -9568.075} C_VEL
LIN {X 0,Y 432.601,Z 394.16,A -85,B 0,C 180,E1 -9569.435,E2 -9569.435} C_VEL
LIN {X 0,Y 432.228,Z 399.907,A -85,B 0,C 180,E1 -9570.889,E2 -9570.889} C_VEL
LIN {X 0,Y 431.844,Z 404.756,A -85,B 0,C 180,E1 -9572.483,E2 -9572.483} C_VEL
LIN {X 0,Y 431.646,Z 407.84,A -85,B 0,C 180,E1 -9573.863,E2 -9573.863} C_VEL
LIN {X 0,Y 431.442,Z 410.235,A -85,B 0,C 180,E1 -9575.465,E2 -9575.465} C_VEL
LIN {X 0,Y 431.353,Z 411.427,A -85,B 0,C 180,E1 -9577.073,E2 -9577.073} C_VEL
LIN {X 0,Y 431.349,Z 411.461,A -85,B 0,C 180,E1 -9578.55,E2 -9578.55} C_VEL
LIN {X 0,Y 431.363,Z 410.496,A -85,B 0,C 180,E1 -9580.027,E2 -9580.027} C_VEL
LIN {X 0,Y 431.516,Z 407.807,A -85,B 0,C 180,E1 -9581.894,E2 -9581.894} C_VEL
LIN {X 0,Y 431.713,Z 405.089,A -85,B 0,C 180,E1 -9583.136,E2 -9583.136} C_VEL
LIN {X 0,Y 431.957,Z 400.416,A -85,B 0,C 180,E1 -9584.709,E2 -9584.709} C_VEL
LIN {X 0,Y 432.274,Z 394.085,A -85,B 0,C 180,E1 -9586.327,E2 -9586.327} C_VEL
LIN {X 0,Y 432.666,Z 387.652,A -85,B 0,C 180,E1 -9587.628,E2 -9587.628} C_VEL
LIN {X 0,Y 433.19,Z 379.688,A -85,B 0,C 180,E1 -9588.94,E2 -9588.94} C_VEL
LIN {X 0,Y 433.759,Z 370.137,A -85,B 0,C 180,E1 -9590.208,E2 -9590.208} C_VEL
LIN {X 0,Y 434.325,Z 359.514,A -85,B 0,C 180,E1 -9591.35,E2 -9591.35} C_VEL
LIN {X 0,Y 434.903,Z 348.798,A -85,B 0,C 180,E1 -9592.266,E2 -9592.266} C_VEL
LIN {X 0,Y 435.452,Z 337.238,A -85,B 0,C 180,E1 -9593.044,E2 -9593.044} C_VEL
LIN {X 0,Y 435.841,Z 325.26,A -85,B 0,C 180,E1 -9593.661,E2 -9593.661} C_VEL
LIN {X 0,Y 436.11,Z 313.214,A -85,B 0,C 180,E1 -9594.106,E2 -9594.106} C_VEL
LIN {X 0,Y 436.3,Z 299.256,A -85,B 0,C 180,E1 -9594.419,E2 -9594.419} C_VEL
LIN {X 0,Y 437.261,Z 216.037,A -85,B 0,C 180,E1 -9595.879,E2 -9595.879} C_VEL
LIN {X 0,Y 432.403,Z 200.624,A -85,B 0,C 180,E1 -9596.377,E2 -9596.377} C_VEL
LIN {X 0,Y 432.333,Z 200.628,A -85,B 0,C 180,E1 -9599.945,E2 -9599.945} C_VEL
LIN {X 0,Y 431.656,Z 200.718,A -85,B 0,C 180,E1 -9600.723,E2 -9600.723} C_VEL
LIN {X 0,Y 428.826,Z 201.065,A -85,B 0,C 180,E1 -9601.988,E2 -9601.988} C_VEL
LIN {X 0,Y 426.431,Z 201.368,A -85,B 0,C 180,E1 -9603.009,E2 -9603.009} C_VEL
LIN {X 0,Y 425.388,Z 201.494,A -85,B 0,C 180,E1 -9603.797,E2 -9603.797} C_VEL
LIN {X 0,Y 425.294,Z 201.504,A -85,B 0,C 180,E1 -9604.064,E2 -9604.064} C_VEL
LIN {X 0,Y 425.284,Z 201.508,A -85,B 0,C 180,E1 -9606.634,E2 -9606.634} C_VEL
LIN {X 0,Y 425.296,Z 201.505,A -85,B 0,C 180,E1 -9609.695,E2 -9609.695} C_VEL
LIN {X 0,Y 425.333,Z 201.504,A -85,B 0,C 180,E1 -9612.697,E2 -9612.697} C_VEL
LIN {X 0,Y 425.348,Z 201.498,A -85,B 0,C 180,E1 -9615.65,E2 -9615.65} C_VEL
LIN {X 0,Y 425.351,Z 201.502,A -85,B 0,C 180,E1 -9618.564,E2 -9618.564} C_VEL
LIN {X 0,Y 425.409,Z 201.491,A -85,B 0,C 180,E1 -9621.45,E2 -9621.45} C_VEL
LIN {X 0,Y 425.542,Z 201.477,A -85,B 0,C 180,E1 -9624.313,E2 -9624.313} C_VEL
LIN {X 0,Y 425.573,Z 201.472,A -85,B 0,C 180,E1 -9628.108,E2 -9628.108} C_VEL
LIN {X 0,Y 425.699,Z 201.456,A -85,B 0,C 180,E1 -9630,E2 -9630} C_VEL
LIN {X 0,Y 425.534,Z 201.477,A -85,B 0,C 180,E1 -9632.84,E2 -9632.84} C_VEL
LIN {X 0,Y 425.542,Z 201.474,A -85,B 0,C 180,E1 -9635.687,E2 -9635.687} C_VEL
LIN {X 0,Y 425.41,Z 201.494,A -85,B 0,C 180,E1 -9638.551,E2 -9638.551} C_VEL
LIN {X 0,Y 425.414,Z 201.494,A -85,B 0,C 180,E1 -9642.402,E2 -9642.402} C_VEL
LIN {X 0,Y 425.389,Z 201.497,A -85,B 0,C 180,E1 -9646.312,E2 -9646.312} C_VEL
LIN {X 0,Y 425.33,Z 201.503,A -85,B 0,C 180,E1 -9649.636,E2 -9649.636} C_VEL
LIN {X 0,Y 425.29,Z 201.508,A -85,B 0,C 180,E1 -9652.339,E2 -9652.339} C_VEL
LIN {X 0,Y 425.32,Z 201.502,A -85,B 0,C 180,E1 -9654.657,E2 -9654.657} C_VEL
LIN {X 0,Y 425.274,Z 201.511,A -85,B 0,C 180,E1 -9657.563,E2 -9657.563} C_VEL
LIN {X 0,Y 425.292,Z 201.505,A -85,B 0,C 180,E1 -9660.761,E2 -9660.761} C_VEL
LIN {X 0,Y 425.313,Z 201.503,A -85,B 0,C 180,E1 -9664.288,E2 -9664.288} C_VEL
LIN {X 0,Y 425.277,Z 201.513,A -85,B 0,C 180,E1 -9667.695,E2 -9667.695} C_VEL
LIN {X 0,Y 425.258,Z 201.509,A -85,B 0,C 180,E1 -9670.517,E2 -9670.517} C_VEL
LIN {X 0,Y 425.258,Z 201.515,A -85,B 0,C 180,E1 -9673.351,E2 -9673.351} C_VEL
LIN {X 0,Y 425.262,Z 201.509,A -85,B 0,C 180,E1 -9676.044,E2 -9676.044} C_VEL
LIN {X 0,Y 425.258,Z 201.509,A -85,B 0,C 180,E1 -9678.619,E2 -9678.619} C_VEL
LIN {X 0,Y 425.283,Z 201.511,A -85,B 0,C 180,E1 -9681.1,E2 -9681.1} C_VEL
LIN {X 0,Y 425.3,Z 201.505,A -85,B 0,C 180,E1 -9684.664,E2 -9684.664} C_VEL
LIN {X 0,Y 425.266,Z 201.508,A -85,B 0,C 180,E1 -9688.073,E2 -9688.073} C_VEL
LIN {X 0,Y 425.308,Z 201.506,A -85,B 0,C 180,E1 -9691.366,E2 -9691.366} C_VEL
LIN {X 0,Y 425.272,Z 201.51,A -85,B 0,C 180,E1 -9694.553,E2 -9694.553} C_VEL
LIN {X 0,Y 425.286,Z 201.509,A -85,B 0,C 180,E1 -9696.634,E2 -9696.634} C_VEL
LIN {X 0,Y 425.298,Z 201.504,A -85,B 0,C 180,E1 -9699.695,E2 -9699.695} C_VEL
LIN {X 0,Y 425.335,Z 201.506,A -85,B 0,C 180,E1 -9702.697,E2 -9702.697} C_VEL
LIN {X 0,Y 425.347,Z 201.498,A -85,B 0,C 180,E1 -9705.65,E2 -9705.65} C_VEL
LIN {X 0,Y 425.353,Z 201.504,A -85,B 0,C 180,E1 -9708.564,E2 -9708.564} C_VEL
LIN {X 0,Y 425.411,Z 201.49,A -85,B 0,C 180,E1 -9711.449,E2 -9711.449} C_VEL
LIN {X 0,Y 425.534,Z 201.48,A -85,B 0,C 180,E1 -9714.313,E2 -9714.313} C_VEL
LIN {X 0,Y 425.574,Z 201.473,A -85,B 0,C 180,E1 -9718.107,E2 -9718.107} C_VEL
LIN {X 0,Y 425.614,Z 201.468,A -85,B 0,C 180,E1 -9720,E2 -9720} C_VEL
LIN {X 0,Y 425.518,Z 201.478,A -85,B 0,C 180,E1 -9722.84,E2 -9722.84} C_VEL
LIN {X 0,Y 425.53,Z 201.477,A -85,B 0,C 180,E1 -9725.687,E2 -9725.687} C_VEL
LIN {X 0,Y 425.41,Z 201.493,A -85,B 0,C 180,E1 -9728.551,E2 -9728.551} C_VEL
LIN {X 0,Y 425.415,Z 201.493,A -85,B 0,C 180,E1 -9732.402,E2 -9732.402} C_VEL
LIN {X 0,Y 425.307,Z 201.504,A -85,B 0,C 180,E1 -9735.331,E2 -9735.331} C_VEL
LIN {X 0,Y 425.316,Z 201.505,A -85,B 0,C 180,E1 -9738.298,E2 -9738.298} C_VEL
LIN {X 0,Y 425.296,Z 201.506,A -85,B 0,C 180,E1 -9741.318,E2 -9741.318} C_VEL
LIN {X 0,Y 425.303,Z 201.503,A -85,B 0,C 180,E1 -9744.651,E2 -9744.651} C_VEL
LIN {X 0,Y 425.254,Z 201.515,A -85,B 0,C 180,E1 -9747.565,E2 -9747.565} C_VEL
LIN {X 0,Y 425.293,Z 201.505,A -85,B 0,C 180,E1 -9750.761,E2 -9750.761} C_VEL
LIN {X 0,Y 425.294,Z 201.505,A -85,B 0,C 180,E1 -9754.284,E2 -9754.284} C_VEL
LIN {X 0,Y 425.278,Z 201.511,A -85,B 0,C 180,E1 -9757.695,E2 -9757.695} C_VEL
LIN {X 0,Y 425.246,Z 201.51,A -85,B 0,C 180,E1 -9760.514,E2 -9760.514} C_VEL
LIN {X 0,Y 425.249,Z 201.517,A -85,B 0,C 180,E1 -9763.349,E2 -9763.349} C_VEL
LIN {X 0,Y 425.259,Z 201.509,A -85,B 0,C 180,E1 -9766.043,E2 -9766.043} C_VEL
LIN {X 0,Y 425.255,Z 201.513,A -85,B 0,C 180,E1 -9769.484,E2 -9769.484} C_VEL
LIN {X 0,Y 425.278,Z 201.507,A -85,B 0,C 180,E1 -9772.489,E2 -9772.489} C_VEL
LIN {X 0,Y 425.288,Z 201.506,A -85,B 0,C 180,E1 -9775.815,E2 -9775.815} C_VEL
LIN {X 0,Y 425.291,Z 201.511,A -85,B 0,C 180,E1 -9779.239,E2 -9779.239} C_VEL
LIN {X 0,Y 425.362,Z 201.561,A -85,B 0,C 180,E1 -9780.862,E2 -9780.862} C_VEL
LIN {X 0,Y 428.592,Z 217.634,A -85,B 0,C 180,E1 -9783.923,E2 -9783.923} C_VEL
LIN {X 0,Y 428.216,Z 226.778,A -85,B 0,C 180,E1 -9785.518,E2 -9785.518} C_VEL
LIN {X 0,Y 427.15,Z 245.768,A -85,B 0,C 180,E1 -9788.778,E2 -9788.778} C_VEL
LIN {X 0,Y 426.321,Z 261.035,A -85,B 0,C 180,E1 -9791.373,E2 -9791.373} C_VEL
LIN {X 0,Y 429.97,Z 290.343,A -85,B 0,C 180,E1 -9792.082,E2 -9792.082} C_VEL
LIN {X 0,Y 428.977,Z 370.184,A -85,B 0,C 180,E1 -9793.523,E2 -9793.523} C_VEL
LIN {X 0,Y 428.524,Z 383.276,A -85,B 0,C 180,E1 -9793.933,E2 -9793.933} C_VEL
LIN {X 0,Y 427.902,Z 395.98,A -85,B 0,C 180,E1 -9794.52,E2 -9794.52} C_VEL
LIN {X 0,Y 427.244,Z 407.347,A -85,B 0,C 180,E1 -9795.228,E2 -9795.228} C_VEL
LIN {X 0,Y 426.472,Z 419.091,A -85,B 0,C 180,E1 -9796.175,E2 -9796.175} C_VEL
LIN {X 0,Y 425.932,Z 428.996,A -85,B 0,C 180,E1 -9797.173,E2 -9797.173} C_VEL
LIN {X 0,Y 425.442,Z 438.357,A -85,B 0,C 180,E1 -9798.325,E2 -9798.325} C_VEL
LIN {X 0,Y 424.888,Z 446.336,A -85,B 0,C 180,E1 -9799.516,E2 -9799.516} C_VEL
LIN {X 0,Y 424.563,Z 454.131,A -85,B 0,C 180,E1 -9800.952,E2 -9800.952} C_VEL
LIN {X 0,Y 424.355,Z 460.384,A -85,B 0,C 180,E1 -9802.386,E2 -9802.386} C_VEL
LIN {X 0,Y 424.216,Z 465.966,A -85,B 0,C 180,E1 -9804.027,E2 -9804.027} C_VEL
LIN {X 0,Y 424.234,Z 469.123,A -85,B 0,C 180,E1 -9805.248,E2 -9805.248} C_VEL
LIN {X 0,Y 424.243,Z 471.069,A -85,B 0,C 180,E1 -9806.2,E2 -9806.2} C_VEL
LIN {X 0,Y 424.315,Z 472.573,A -85,B 0,C 180,E1 -9807.152,E2 -9807.152} C_VEL
LIN {X 0,Y 424.337,Z 473.609,A -85,B 0,C 180,E1 -9808.101,E2 -9808.101} C_VEL
LIN {X 0,Y 424.275,Z 474.235,A -85,B 0,C 180,E1 -9809.051,E2 -9809.051} C_VEL
LIN {X 0,Y 424.255,Z 474.463,A -85,B 0,C 180,E1 -9810,E2 -9810} C_VEL
LIN {X 0,Y 424.275,Z 474.268,A -85,B 0,C 180,E1 -9810.949,E2 -9810.949} C_VEL
LIN {X 0,Y 424.31,Z 473.636,A -85,B 0,C 180,E1 -9811.898,E2 -9811.898} C_VEL
LIN {X 0,Y 424.32,Z 472.601,A -85,B 0,C 180,E1 -9812.848,E2 -9812.848} C_VEL
LIN {X 0,Y 424.248,Z 471.15,A -85,B 0,C 180,E1 -9813.799,E2 -9813.799} C_VEL
LIN {X 0,Y 424.261,Z 468.116,A -85,B 0,C 180,E1 -9815.227,E2 -9815.227} C_VEL
LIN {X 0,Y 424.299,Z 464.018,A -85,B 0,C 180,E1 -9816.658,E2 -9816.658} C_VEL
LIN {X 0,Y 424.484,Z 457.745,A -85,B 0,C 180,E1 -9818.33,E2 -9818.33} C_VEL
LIN {X 0,Y 424.738,Z 450.897,A -85,B 0,C 180,E1 -9819.765,E2 -9819.765} C_VEL
LIN {X 0,Y 425.238,Z 442.43,A -85,B 0,C 180,E1 -9821.197,E2 -9821.197} C_VEL
LIN {X 0,Y 425.699,Z 433.776,A -85,B 0,C 180,E1 -9822.393,E2 -9822.393} C_VEL
LIN {X 0,Y 426.385,Z 423.361,A -85,B 0,C 180,E1 -9823.56,E2 -9823.56} C_VEL
LIN {X 0,Y 427.126,Z 412.616,A -85,B 0,C 180,E1 -9824.532,E2 -9824.532} C_VEL
LIN {X 0,Y 427.895,Z 401.151,A -85,B 0,C 180,E1 -9825.358,E2 -9825.358} C_VEL
LIN {X 0,Y 428.579,Z 389.449,A -85,B 0,C 180,E1 -9826.003,E2 -9826.003} C_VEL
LIN {X 0,Y 429.23,Z 376.158,A -85,B 0,C 180,E1 -9826.528,E2 -9826.528} C_VEL
LIN {X 0,Y 429.649,Z 363.467,A -85,B 0,C 180,E1 -9826.848,E2 -9826.848} C_VEL
LIN {X 0,Y 430.445,Z 288.37,A -85,B 0,C 180,E1 -9828.22,E2 -9828.22} C_VEL
LIN {X 0,Y 427.485,Z 265.341,A -85,B 0,C 180,E1 -9828.81,E2 -9828.81} C_VEL
LIN {X 0,Y 426.439,Z 258.592,A -85,B 0,C 180,E1 -9829.005,E2 -9829.005} C_VEL
LIN {X 0,Y 427.269,Z 240.62,A -85,B 0,C 180,E1 -9831.975,E2 -9831.975} C_VEL
LIN {X 0,Y 428.315,Z 221.066,A -85,B 0,C 180,E1 -9835.253,E2 -9835.253} C_VEL
LIN {X 0,Y 428.397,Z 216.304,A -85,B 0,C 180,E1 -9836.068,E2 -9836.068} C_VEL
LIN {X 0,Y 425.928,Z 204.243,A -85,B 0,C 180,E1 -9838.319,E2 -9838.319} C_VEL
LIN {X 0,Y 425.306,Z 201.513,A -85,B 0,C 180,E1 -9838.859,E2 -9838.859} C_VEL
LIN {X 0,Y 425.264,Z 201.513,A -85,B 0,C 180,E1 -9841.927,E2 -9841.927} C_VEL
LIN {X 0,Y 425.298,Z 201.507,A -85,B 0,C 180,E1 -9845.336,E2 -9845.336} C_VEL
LIN {X 0,Y 425.28,Z 201.51,A -85,B 0,C 180,E1 -9848.9,E2 -9848.9} C_VEL
LIN {X 0,Y 425.269,Z 201.511,A -85,B 0,C 180,E1 -9852.653,E2 -9852.653} C_VEL
LIN {X 0,Y 425.261,Z 201.51,A -85,B 0,C 180,E1 -9856.044,E2 -9856.044} C_VEL
LIN {X 0,Y 425.258,Z 201.515,A -85,B 0,C 180,E1 -9858.619,E2 -9858.619} C_VEL
LIN {X 0,Y 425.28,Z 201.509,A -85,B 0,C 180,E1 -9861.099,E2 -9861.099} C_VEL
LIN {X 0,Y 425.299,Z 201.506,A -85,B 0,C 180,E1 -9864.664,E2 -9864.664} C_VEL
LIN {X 0,Y 425.265,Z 201.511,A -85,B 0,C 180,E1 -9868.073,E2 -9868.073} C_VEL
LIN {X 0,Y 425.314,Z 201.502,A -85,B 0,C 180,E1 -9871.366,E2 -9871.366} C_VEL
LIN {X 0,Y 425.271,Z 201.511,A -85,B 0,C 180,E1 -9874.553,E2 -9874.553} C_VEL
LIN {X 0,Y 425.283,Z 201.507,A -85,B 0,C 180,E1 -9876.633,E2 -9876.633} C_VEL
LIN {X 0,Y 425.295,Z 201.507,A -85,B 0,C 180,E1 -9879.694,E2 -9879.694} C_VEL
LIN {X 0,Y 425.332,Z 201.498,A -85,B 0,C 180,E1 -9882.697,E2 -9882.697} C_VEL
LIN {X 0,Y 425.346,Z 201.5,A -85,B 0,C 180,E1 -9885.65,E2 -9885.65} C_VEL
LIN {X 0,Y 425.35,Z 201.496,A -85,B 0,C 180,E1 -9888.564,E2 -9888.564} C_VEL
LIN {X 0,Y 425.538,Z 201.476,A -85,B 0,C 180,E1 -9892.408,E2 -9892.408} C_VEL
LIN {X 0,Y 425.55,Z 201.474,A -85,B 0,C 180,E1 -9894.313,E2 -9894.313} C_VEL
LIN {X 0,Y 425.572,Z 201.471,A -85,B 0,C 180,E1 -9898.107,E2 -9898.107} C_VEL
LIN {X 0,Y 425.702,Z 201.457,A -85,B 0,C 180,E1 -9900,E2 -9900} C_VEL
LIN {X 0,Y 425.546,Z 201.478,A -85,B 0,C 180,E1 -9902.84,E2 -9902.84} C_VEL
LIN {X 0,Y 425.498,Z 201.482,A -85,B 0,C 180,E1 -9906.504,E2 -9906.504} C_VEL
LIN {X 0,Y 425.398,Z 201.499,A -85,B 0,C 180,E1 -9909.509,E2 -9909.509} C_VEL
LIN {X 0,Y 425.393,Z 201.502,A -85,B 0,C 180,E1 -9912.904,E2 -9912.904} C_VEL
LIN {X 0,Y 425.38,Z 201.5,A -85,B 0,C 180,E1 -9916.613,E2 -9916.613} C_VEL
LIN {X 0,Y 425.374,Z 201.626,A -85,B 0,C 180,E1 -9918.763,E2 -9918.763} C_VEL
LIN {X 0,Y 425.712,Z 202.994,A -85,B 0,C 180,E1 -9919.029,E2 -9919.029} C_VEL
LIN {X 0,Y 431.514,Z 218.359,A -85,B 0,C 180,E1 -9919.636,E2 -9919.636} C_VEL
LIN {X 0,Y 430.061,Z 309.954,A -85,B 0,C 180,E1 -9921.333,E2 -9921.333} C_VEL
LIN {X 0,Y 429.744,Z 322.294,A -85,B 0,C 180,E1 -9921.727,E2 -9921.727} C_VEL
LIN {X 0,Y 429.324,Z 334.702,A -85,B 0,C 180,E1 -9922.307,E2 -9922.307} C_VEL
LIN {X 0,Y 428.809,Z 346.296,A -85,B 0,C 180,E1 -9923.035,E2 -9923.035} C_VEL
LIN {X 0,Y 428.174,Z 357.842,A -85,B 0,C 180,E1 -9923.979,E2 -9923.979} C_VEL
LIN {X 0,Y 427.509,Z 367.979,A -85,B 0,C 180,E1 -9925.015,E2 -9925.015} C_VEL
LIN {X 0,Y 426.936,Z 376.829,A -85,B 0,C 180,E1 -9926.126,E2 -9926.126} C_VEL
LIN {X 0,Y 426.289,Z 385.683,A -85,B 0,C 180,E1 -9927.492,E2 -9927.492} C_VEL
LIN {X 0,Y 425.737,Z 393.297,A -85,B 0,C 180,E1 -9928.965,E2 -9928.965} C_VEL
LIN {X 0,Y 425.336,Z 398.565,A -85,B 0,C 180,E1 -9930.227,E2 -9930.227} C_VEL
LIN {X 0,Y 424.906,Z 404.225,A -85,B 0,C 180,E1 -9931.957,E2 -9931.957} C_VEL
LIN {X 0,Y 424.604,Z 408.096,A -85,B 0,C 180,E1 -9933.616,E2 -9933.616} C_VEL
LIN {X 0,Y 424.388,Z 410.795,A -85,B 0,C 180,E1 -9935.423,E2 -9935.423} C_VEL
LIN {X 0,Y 424.26,Z 412.045,A -85,B 0,C 180,E1 -9937.332,E2 -9937.332} C_VEL
LIN {X 0,Y 424.287,Z 411.78,A -85,B 0,C 180,E1 -9939.009,E2 -9939.009} C_VEL
LIN {X 0,Y 424.288,Z 410.676,A -85,B 0,C 180,E1 -9940.364,E2 -9940.364} C_VEL
LIN {X 0,Y 424.447,Z 408.519,A -85,B 0,C 180,E1 -9941.832,E2 -9941.832} C_VEL
LIN {X 0,Y 424.721,Z 404.515,A -85,B 0,C 180,E1 -9943.605,E2 -9943.605} C_VEL
LIN {X 0,Y 425.043,Z 399.106,A -85,B 0,C 180,E1 -9945.316,E2 -9945.316} C_VEL
LIN {X 0,Y 425.32,Z 393.697,A -85,B 0,C 180,E1 -9946.64,E2 -9946.64} C_VEL
LIN {X 0,Y 425.809,Z 385.864,A -85,B 0,C 180,E1 -9948.167,E2 -9948.167} C_VEL
LIN {X 0,Y 426.388,Z 377.392,A -85,B 0,C 180,E1 -9949.495,E2 -9949.495} C_VEL
LIN {X 0,Y 426.972,Z 368.1,A -85,B 0,C 180,E1 -9950.681,E2 -9950.681} C_VEL
LIN {X 0,Y 427.543,Z 356.818,A -85,B 0,C 180,E1 -9951.834,E2 -9951.834} C_VEL
LIN {X 0,Y 428.163,Z 346.001,A -85,B 0,C 180,E1 -9952.713,E2 -9952.713} C_VEL
LIN {X 0,Y 428.7,Z 334.529,A -85,B 0,C 180,E1 -9953.446,E2 -9953.446} C_VEL
LIN {X 0,Y 429.012,Z 321.173,A -85,B 0,C 180,E1 -9954.077,E2 -9954.077} C_VEL
LIN {X 0,Y 429.306,Z 307.631,A -85,B 0,C 180,E1 -9954.501,E2 -9954.501} C_VEL
LIN {X 0,Y 430.486,Z 217.144,A -85,B 0,C 180,E1 -9956.131,E2 -9956.131} C_VEL
LIN {X 0,Y 425.329,Z 201.505,A -85,B 0,C 180,E1 -9956.656,E2 -9956.656} C_VEL
LIN {X 0,Y 425.291,Z 201.505,A -85,B 0,C 180,E1 -9960.281,E2 -9960.281} C_VEL
LIN {X 0,Y 425.346,Z 201.501,A -85,B 0,C 180,E1 -9963.505,E2 -9963.505} C_VEL
LIN {X 0,Y 425.294,Z 201.504,A -85,B 0,C 180,E1 -9964.064,E2 -9964.064} C_VEL
LIN {X 0,Y 424.598,Z 201.597,A -85,B 0,C 180,E1 -9964.854,E2 -9964.854} C_VEL
LIN {X 0,Y 421.72,Z 201.95,A -85,B 0,C 180,E1 -9966.138,E2 -9966.138} C_VEL
LIN {X 0,Y 419.315,Z 202.255,A -85,B 0,C 180,E1 -9967.174,E2 -9967.174} C_VEL
LIN {X 0,Y 418.303,Z 202.376,A -85,B 0,C 180,E1 -9967.975,E2 -9967.975} C_VEL
LIN {X 0,Y 418.232,Z 202.385,A -85,B 0,C 180,E1 -9968.246,E2 -9968.246} C_VEL
LIN {X 0,Y 418.276,Z 202.381,A -85,B 0,C 180,E1 -9971.383,E2 -9971.383} C_VEL
LIN {X 0,Y 418.302,Z 202.378,A -85,B 0,C 180,E1 -9974.406,E2 -9974.406} C_VEL
LIN {X 0,Y 418.357,Z 202.37,A -85,B 0,C 180,E1 -9977.386,E2 -9977.386} C_VEL
LIN {X 0,Y 418.34,Z 202.373,A -85,B 0,C 180,E1 -9980.329,E2 -9980.329} C_VEL
LIN {X 0,Y 418.461,Z 202.357,A -85,B 0,C 180,E1 -9983.249,E2 -9983.249} C_VEL
LIN {X 0,Y 418.334,Z 202.373,A -85,B 0,C 180,E1 -9985.182,E2 -9985.182} C_VEL
LIN {X 0,Y 418.542,Z 202.348,A -85,B 0,C 180,E1 -9988.076,E2 -9988.076} C_VEL
LIN {X 0,Y 418.668,Z 202.332,A -85,B 0,C 180,E1 -9990,E2 -9990} C_VEL
LIN {X 0,Y 418.489,Z 202.354,A -85,B 0,C 180,E1 -9992.888,E2 -9992.888} C_VEL
LIN {X 0,Y 418.5,Z 202.352,A -85,B 0,C 180,E1 -9995.783,E2 -9995.783} C_VEL
LIN {X 0,Y 418.379,Z 202.369,A -85,B 0,C 180,E1 -9998.696,E2 -9998.696} C_VEL
LIN {X 0,Y 418.316,Z 202.375,A -85,B 0,C 180,E1 -10001.631,E2 -10001.631} C_VEL
LIN {X 0,Y 418.303,Z 202.378,A -85,B 0,C 180,E1 -10004.597,E2 -10004.597} C_VEL
LIN {X 0,Y 418.287,Z 202.379,A -85,B 0,C 180,E1 -10007.604,E2 -10007.604} C_VEL
LIN {X 0,Y 418.252,Z 202.383,A -85,B 0,C 180,E1 -10010.663,E2 -10010.663} C_VEL
LIN {X 0,Y 418.275,Z 202.384,A -85,B 0,C 180,E1 -10013.782,E2 -10013.782} C_VEL
LIN {X 0,Y 418.228,Z 202.385,A -85,B 0,C 180,E1 -10017.048,E2 -10017.048} C_VEL
LIN {X 0,Y 418.244,Z 202.385,A -85,B 0,C 180,E1 -10020.272,E2 -10020.272} C_VEL
LIN {X 0,Y 418.25,Z 202.389,A -85,B 0,C 180,E1 -10023.677,E2 -10023.677} C_VEL
LIN {X 0,Y 418.24,Z 202.386,A -85,B 0,C 180,E1 -10027.225,E2 -10027.225} C_VEL
LIN {X 0,Y 418.214,Z 202.387,A -85,B 0,C 180,E1 -10030.868,E2 -10030.868} C_VEL
LIN {X 0,Y 418.211,Z 202.391,A -85,B 0,C 180,E1 -10033.729,E2 -10033.729} C_VEL
LIN {X 0,Y 418.209,Z 202.387,A -85,B 0,C 180,E1 -10036.449,E2 -10036.449} C_VEL
LIN {X 0,Y 418.211,Z 202.392,A -85,B 0,C 180,E1 -10039.133,E2 -10039.133} C_VEL
LIN {X 0,Y 418.241,Z 202.385,A -85,B 0,C 180,E1 -10042.776,E2 -10042.776} C_VEL
LIN {X 0,Y 418.25,Z 202.382,A -85,B 0,C 180,E1 -10046.323,E2 -10046.323} C_VEL
LIN {X 0,Y 418.244,Z 202.384,A -85,B 0,C 180,E1 -10049.728,E2 -10049.728} C_VEL
LIN {X 0,Y 418.227,Z 202.392,A -85,B 0,C 180,E1 -10053.018,E2 -10053.018} C_VEL
LIN {X 0,Y 418.276,Z 202.379,A -85,B 0,C 180,E1 -10056.218,E2 -10056.218} C_VEL
LIN {X 0,Y 418.253,Z 202.384,A -85,B 0,C 180,E1 -10059.337,E2 -10059.337} C_VEL
LIN {X 0,Y 418.282,Z 202.381,A -85,B 0,C 180,E1 -10062.396,E2 -10062.396} C_VEL
LIN {X 0,Y 418.303,Z 202.376,A -85,B 0,C 180,E1 -10065.403,E2 -10065.403} C_VEL
LIN {X 0,Y 418.317,Z 202.378,A -85,B 0,C 180,E1 -10068.369,E2 -10068.369} C_VEL
LIN {X 0,Y 418.38,Z 202.366,A -85,B 0,C 180,E1 -10071.305,E2 -10071.305} C_VEL
LIN {X 0,Y 418.492,Z 202.356,A -85,B 0,C 180,E1 -10074.217,E2 -10074.217} C_VEL
LIN {X 0,Y 418.543,Z 202.349,A -85,B 0,C 180,E1 -10078.076,E2 -10078.076} C_VEL
LIN {X 0,Y 418.468,Z 202.356,A -85,B 0,C 180,E1 -10080.962,E2 -10080.962} C_VEL
LIN {X 0,Y 418.475,Z 202.355,A -85,B 0,C 180,E1 -10082.888,E2 -10082.888} C_VEL
LIN {X 0,Y 418.487,Z 202.355,A -85,B 0,C 180,E1 -10085.783,E2 -10085.783} C_VEL
LIN {X 0,Y 418.379,Z 202.367,A -85,B 0,C 180,E1 -10088.696,E2 -10088.696} C_VEL
LIN {X 0,Y 418.317,Z 202.376,A -85,B 0,C 180,E1 -10091.631,E2 -10091.631} C_VEL
LIN {X 0,Y 418.282,Z 202.379,A -85,B 0,C 180,E1 -10094.598,E2 -10094.598} C_VEL
LIN {X 0,Y 418.259,Z 202.384,A -85,B 0,C 180,E1 -10097.605,E2 -10097.605} C_VEL
LIN {X 0,Y 418.253,Z 202.382,A -85,B 0,C 180,E1 -10100.663,E2 -10100.663} C_VEL
LIN {X 0,Y 418.262,Z 202.388,A -85,B 0,C 180,E1 -10103.783,E2 -10103.783} C_VEL
LIN {X 0,Y 418.211,Z 202.387,A -85,B 0,C 180,E1 -10107.043,E2 -10107.043} C_VEL
LIN {X 0,Y 418.244,Z 202.384,A -85,B 0,C 180,E1 -10110.272,E2 -10110.272} C_VEL
LIN {X 0,Y 418.235,Z 202.39,A -85,B 0,C 180,E1 -10113.679,E2 -10113.679} C_VEL
LIN {X 0,Y 418.241,Z 202.387,A -85,B 0,C 180,E1 -10117.224,E2 -10117.224} C_VEL
LIN {X 0,Y 418.209,Z 202.389,A -85,B 0,C 180,E1 -10120.867,E2 -10120.867} C_VEL
LIN {X 0,Y 418.205,Z 202.39,A -85,B 0,C 180,E1 -10123.728,E2 -10123.728} C_VEL
LIN {X 0,Y 418.202,Z 202.388,A -85,B 0,C 180,E1 -10126.447,E2 -10126.447} C_VEL
LIN {X 0,Y 418.212,Z 202.393,A -85,B 0,C 180,E1 -10129.132,E2 -10129.132} C_VEL
LIN {X 0,Y 418.241,Z 202.386,A -85,B 0,C 180,E1 -10132.775,E2 -10132.775} C_VEL
LIN {X 0,Y 418.235,Z 202.384,A -85,B 0,C 180,E1 -10136.321,E2 -10136.321} C_VEL
LIN {X 0,Y 418.249,Z 202.385,A -85,B 0,C 180,E1 -10139.728,E2 -10139.728} C_VEL
LIN {X 0,Y 418.293,Z 202.525,A -85,B 0,C 180,E1 -10140.633,E2 -10140.633} C_VEL
LIN {X 0,Y 421.341,Z 217.222,A -85,B 0,C 180,E1 -10143.491,E2 -10143.491} C_VEL
LIN {X 0,Y 421.728,Z 220.741,A -85,B 0,C 180,E1 -10144.145,E2 -10144.145} C_VEL
LIN {X 0,Y 420.567,Z 239.283,A -85,B 0,C 180,E1 -10147.396,E2 -10147.396} C_VEL
LIN {X 0,Y 419.514,Z 258.214,A -85,B 0,C 180,E1 -10150.678,E2 -10150.678} C_VEL
LIN {X 0,Y 419.367,Z 260.573,A -85,B 0,C 180,E1 -10151.084,E2 -10151.084} C_VEL
LIN {X 0,Y 423.131,Z 290.012,A -85,B 0,C 180,E1 -10151.814,E2 -10151.814} C_VEL
LIN {X 0,Y 422.086,Z 370.603,A -85,B 0,C 180,E1 -10153.308,E2 -10153.308} C_VEL
LIN {X 0,Y 421.589,Z 384.144,A -85,B 0,C 180,E1 -10153.755,E2 -10153.755} C_VEL
LIN {X 0,Y 420.904,Z 396.99,A -85,B 0,C 180,E1 -10154.38,E2 -10154.38} C_VEL
LIN {X 0,Y 420.117,Z 409.562,A -85,B 0,C 180,E1 -10155.219,E2 -10155.219} C_VEL
LIN {X 0,Y 419.351,Z 420.817,A -85,B 0,C 180,E1 -10156.183,E2 -10156.183} C_VEL
LIN {X 0,Y 418.84,Z 430.413,A -85,B 0,C 180,E1 -10157.207,E2 -10157.207} C_VEL
LIN {X 0,Y 418.332,Z 439.336,A -85,B 0,C 180,E1 -10158.369,E2 -10158.369} C_VEL
LIN {X 0,Y 417.708,Z 448.426,A -85,B 0,C 180,E1 -10159.824,E2 -10159.824} C_VEL
LIN {X 0,Y 417.428,Z 455.751,A -85,B 0,C 180,E1 -10161.284,E2 -10161.284} C_VEL
LIN {X 0,Y 417.254,Z 461.578,A -85,B 0,C 180,E1 -10162.742,E2 -10162.742} C_VEL
LIN {X 0,Y 417.141,Z 466.144,A -85,B 0,C 180,E1 -10164.198,E2 -10164.198} C_VEL
LIN {X 0,Y 417.169,Z 468.547,A -85,B 0,C 180,E1 -10165.168,E2 -10165.168} C_VEL
LIN {X 0,Y 417.15,Z 470.5,A -85,B 0,C 180,E1 -10166.136,E2 -10166.136} C_VEL
LIN {X 0,Y 417.242,Z 472.022,A -85,B 0,C 180,E1 -10167.103,E2 -10167.103} C_VEL
LIN {X 0,Y 417.253,Z 473.067,A -85,B 0,C 180,E1 -10168.069,E2 -10168.069} C_VEL
LIN {X 0,Y 417.218,Z 473.702,A -85,B 0,C 180,E1 -10169.035,E2 -10169.035} C_VEL
LIN {X 0,Y 417.197,Z 473.936,A -85,B 0,C 180,E1 -10170,E2 -10170} C_VEL
LIN {X 0,Y 417.218,Z 473.753,A -85,B 0,C 180,E1 -10170.965,E2 -10170.965} C_VEL
LIN {X 0,Y 417.228,Z 473.124,A -85,B 0,C 180,E1 -10171.93,E2 -10171.93} C_VEL
LIN {X 0,Y 417.247,Z 472.094,A -85,B 0,C 180,E1 -10172.896,E2 -10172.896} C_VEL
LIN {X 0,Y 417.153,Z 470.647,A -85,B 0,C 180,E1 -10173.864,E2 -10173.864} C_VEL
LIN {X 0,Y 417.168,Z 467.625,A -85,B 0,C 180,E1 -10175.316,E2 -10175.316} C_VEL
LIN {X 0,Y 417.23,Z 463.542,A -85,B 0,C 180,E1 -10176.771,E2 -10176.771} C_VEL
LIN {X 0,Y 417.421,Z 457.292,A -85,B 0,C 180,E1 -10178.471,E2 -10178.471} C_VEL
LIN {X 0,Y 417.668,Z 450.456,A -85,B 0,C 180,E1 -10179.931,E2 -10179.931} C_VEL
LIN {X 0,Y 418.226,Z 442.002,A -85,B 0,C 180,E1 -10181.388,E2 -10181.388} C_VEL
LIN {X 0,Y 418.736,Z 433.372,A -85,B 0,C 180,E1 -10182.602,E2 -10182.602} C_VEL
LIN {X 0,Y 419.484,Z 422.75,A -85,B 0,C 180,E1 -10183.812,E2 -10183.812} C_VEL
LIN {X 0,Y 420.336,Z 410.835,A -85,B 0,C 180,E1 -10184.896,E2 -10184.896} C_VEL
LIN {X 0,Y 421.158,Z 398.958,A -85,B 0,C 180,E1 -10185.734,E2 -10185.734} C_VEL
LIN {X 0,Y 421.861,Z 386.722,A -85,B 0,C 180,E1 -10186.39,E2 -10186.39} C_VEL
LIN {X 0,Y 422.54,Z 373.553,A -85,B 0,C 180,E1 -10186.891,E2 -10186.891} C_VEL
LIN {X 0,Y 422.942,Z 360.996,A -85,B 0,C 180,E1 -10187.185,E2 -10187.185} C_VEL
LIN {X 0,Y 423.816,Z 289.585,A -85,B 0,C 180,E1 -10188.518,E2 -10188.518} C_VEL
LIN {X 0,Y 420.964,Z 267.272,A -85,B 0,C 180,E1 -10189.102,E2 -10189.102} C_VEL
LIN {X 0,Y 419.527,Z 258.011,A -85,B 0,C 180,E1 -10189.365,E2 -10189.365} C_VEL
LIN {X 0,Y 420.487,Z 238.787,A -85,B 0,C 180,E1 -10192.608,E2 -10192.608} C_VEL
LIN {X 0,Y 421.615,Z 219.196,A -85,B 0,C 180,E1 -10195.948,E2 -10195.948} C_VEL
LIN {X 0,Y 420.009,Z 210.099,A -85,B 0,C 180,E1 -10197.658,E2 -10197.658} C_VEL
LIN {X 0,Y 418.259,Z 202.392,A -85,B 0,C 180,E1 -10199.162,E2 -10199.162} C_VEL
LIN {X 0,Y 418.258,Z 202.387,A -85,B 0,C 180,E1 -10202.843,E2 -10202.843} C_VEL
LIN {X 0,Y 418.244,Z 202.385,A -85,B 0,C 180,E1 -10206.237,E2 -10206.237} C_VEL
LIN {X 0,Y 418.201,Z 202.39,A -85,B 0,C 180,E1 -10209.687,E2 -10209.687} C_VEL
LIN {X 0,Y 418.222,Z 202.39,A -85,B 0,C 180,E1 -10212.32,E2 -10212.32} C_VEL
LIN {X 0,Y 418.236,Z 202.385,A -85,B 0,C 180,E1 -10215.108,E2 -10215.108} C_VEL
LIN {X 0,Y 418.232,Z 202.383,A -85,B 0,C 180,E1 -10217.766,E2 -10217.766} C_VEL
LIN {X 0,Y 418.238,Z 202.385,A -85,B 0,C 180,E1 -10221.556,E2 -10221.556} C_VEL
LIN {X 0,Y 418.259,Z 202.381,A -85,B 0,C 180,E1 -10225.159,E2 -10225.159} C_VEL
LIN {X 0,Y 418.245,Z 202.383,A -85,B 0,C 180,E1 -10227.472,E2 -10227.472} C_VEL
LIN {X 0,Y 418.264,Z 202.381,A -85,B 0,C 180,E1 -10230.896,E2 -10230.896} C_VEL
LIN {X 0,Y 418.236,Z 202.387,A -85,B 0,C 180,E1 -10234.094,E2 -10234.094} C_VEL
LIN {X 0,Y 418.231,Z 202.385,A -85,B 0,C 180,E1 -10237.263,E2 -10237.263} C_VEL
LIN {X 0,Y 418.283,Z 202.382,A -85,B 0,C 180,E1 -10240.364,E2 -10240.364} C_VEL
LIN {X 0,Y 418.316,Z 202.375,A -85,B 0,C 180,E1 -10243.404,E2 -10243.404} C_VEL
LIN {X 0,Y 418.346,Z 202.372,A -85,B 0,C 180,E1 -10246.999,E2 -10246.999} C_VEL
LIN {X 0,Y 418.34,Z 202.371,A -85,B 0,C 180,E1 -10250.329,E2 -10250.329} C_VEL
LIN {X 0,Y 418.487,Z 202.358,A -85,B 0,C 180,E1 -10253.249,E2 -10253.249} C_VEL
LIN {X 0,Y 418.336,Z 202.376,A -85,B 0,C 180,E1 -10255.181,E2 -10255.181} C_VEL
LIN {X 0,Y 418.541,Z 202.347,A -85,B 0,C 180,E1 -10258.075,E2 -10258.075} C_VEL
LIN {X 0,Y 418.671,Z 202.333,A -85,B 0,C 180,E1 -10260,E2 -10260} C_VEL
LIN {X 0,Y 418.501,Z 202.355,A -85,B 0,C 180,E1 -10262.888,E2 -10262.888} C_VEL
LIN {X 0,Y 418.459,Z 202.358,A -85,B 0,C 180,E1 -10266.503,E2 -10266.503} C_VEL
LIN {X 0,Y 418.339,Z 202.377,A -85,B 0,C 180,E1 -10269.671,E2 -10269.671} C_VEL
LIN {X 0,Y 418.346,Z 202.38,A -85,B 0,C 180,E1 -10273.001,E2 -10273.001} C_VEL
LIN {X 0,Y 418.346,Z 202.377,A -85,B 0,C 180,E1 -10276.75,E2 -10276.75} C_VEL
LIN {X 0,Y 418.315,Z 202.409,A -85,B 0,C 180,E1 -10278.425,E2 -10278.425} C_VEL
LIN {X 0,Y 418.539,Z 203.407,A -85,B 0,C 180,E1 -10278.637,E2 -10278.637} C_VEL
LIN {X 0,Y 424.865,Z 219.893,A -85,B 0,C 180,E1 -10279.319,E2 -10279.319} C_VEL
LIN {X 0,Y 423.311,Z 311.479,A -85,B 0,C 180,E1 -10281.056,E2 -10281.056} C_VEL
LIN {X 0,Y 423.018,Z 324.615,A -85,B 0,C 180,E1 -10281.506,E2 -10281.506} C_VEL
LIN {X 0,Y 422.54,Z 337.278,A -85,B 0,C 180,E1 -10282.138,E2 -10282.138} C_VEL
LIN {X 0,Y 421.927,Z 348.82,A -85,B 0,C 180,E1 -10282.914,E2 -10282.914} C_VEL
LIN {X 0,Y 421.271,Z 359.863,A -85,B 0,C 180,E1 -10283.864,E2 -10283.864} C_VEL
LIN {X 0,Y 420.588,Z 369.703,A -85,B 0,C 180,E1 -10284.913,E2 -10284.913} C_VEL
LIN {X 0,Y 419.975,Z 378.452,A -85,B 0,C 180,E1 -10286.058,E2 -10286.058} C_VEL
LIN {X 0,Y 419.324,Z 386.487,A -85,B 0,C 180,E1 -10287.34,E2 -10287.34} C_VEL
LIN {X 0,Y 418.76,Z 394.105,A -85,B 0,C 180,E1 -10288.849,E2 -10288.849} C_VEL
